SPLINE
SPL {X  -165.650, Y  +532.042, Z    +0.000, E1   +53.611, E3 +284862.764}
SPL {X  -165.650, Y  +526.147, Z    +0.000, E1   +53.495, E3 +284872.403}
SPL {X  -165.650, Y  +517.365, Z    +0.000, E1   +53.387, E3 +284886.571}
SPL {X  -165.650, Y  +505.685, Z    +0.000, E1   +53.701, E3 +284902.196}
SPL {X  -165.650, Y  +498.275, Z    +0.000, E1   +53.357, E3 +284915.504}
SPL {X  -165.650, Y  +487.031, Z    +0.000, E1   +53.931, E3 +284928.912}
SPL {X  -165.650, Y  +450.615, Z    +0.000, E1   +59.721, E3 +284940.152}
SPL {X  -165.650, Y  +449.326, Z    +0.000, E1   +58.606, E3 +284949.202}
SPL {X  -165.650, Y  +442.154, Z    +0.000, E1   +58.369, E3 +284959.826}
SPL {X  -165.650, Y  +437.405, Z    +0.000, E1   +57.663, E3 +284970.435}
SPL {X  -165.650, Y  +432.227, Z    +0.000, E1   +57.103, E3 +284980.923}
SPL {X  -165.650, Y  +428.683, Z    +0.000, E1   +56.222, E3 +284991.277}
SPL {X  -165.650, Y  +424.202, Z    +0.000, E1   +55.382, E3 +285002.966}
SPL {X  -165.650, Y  +418.469, Z    +0.000, E1   +54.594, E3 +285016.074}
SPL {X  -165.650, Y  +413.857, Z    +0.000, E1   +53.683, E3 +285028.645}
SPL {X  -165.650, Y  +403.104, Z    +0.000, E1   +53.908, E3 +285043.382}
SPL {X  -165.650, Y  +393.046, Z    +0.000, E1   +53.951, E3 +285058.066}
SPL {X  -165.650, Y  +383.306, Z    +0.000, E1   +53.987, E3 +285072.343}
SPL {X  -165.640, Y  +376.676, Z    +0.000, E1   +53.760, E3 +285083.510}
SPL {X  -165.408, Y  +369.556, Z    +0.000, E1   +53.942, E3 +285093.061}
SPL {X  -164.927, Y  +363.041, Z    +0.000, E1   +53.687, E3 +285104.356}
SPL {X  -163.980, Y  +355.035, Z    +0.000, E1   +53.657, E3 +285116.553}
SPL {X  -162.665, Y  +347.197, Z    +0.000, E1   +53.396, E3 +285129.816}
SPL {X  -161.218, Y  +340.437, Z    +0.000, E1   +53.207, E3 +285140.915}
SPL {X  -159.523, Y  +333.864, Z    +0.000, E1   +52.908, E3 +285152.537}
SPL {X  -157.624, Y  +327.563, Z    +0.000, E1   +52.705, E3 +285162.946}
SPL {X  -155.665, Y  +321.859, Z    +0.000, E1   +52.064, E3 +285175.119}
SPL {X  -152.682, Y  +314.249, Z    +0.000, E1   +51.841, E3 +285187.567}
SPL {X  -150.607, Y  +309.525, Z    +0.000, E1   +51.147, E3 +285198.052}
SPL {X  -139.567, Y  +289.276, Z    +0.000, E1   +56.334, E3 +285200.030}
SPL {X  -117.053, Y  +261.289, Z    +0.000, E1   +49.815, E3 +285313.564}
ENDSPLINE

SPLINE
SPL {X  -148.836, Y  +305.783, Z    +0.000, E1   +38.029, E3 +285405.041}
SPL {X  -161.816, Y  +343.065, Z    +0.000, E1   +22.147, E3 +285395.691}
SPL {X  -165.007, Y  +363.921, Z    +0.000, E1   +11.079, E3 +285393.680}
SPL {X  -165.587, Y  +373.939, Z    +0.000, E1    +4.928, E3 +285393.520}
SPL {X  -165.650, Y  +378.704, Z    +0.000, E1    +1.700, E3 +285393.101}
SPL {X  -165.650, Y  +382.197, Z    +0.000, E1    -1.038, E3 +285392.175}
SPL {X  -165.650, Y  +386.782, Z    +0.000, E1    -5.783, E3 +285391.652}
SPL {X  -165.650, Y  +392.406, Z    +0.000, E1   -13.042, E3 +285389.550}
SPL {X  -165.650, Y  +398.038, Z    +0.000, E1   -20.113, E3 +285391.117}
SPL {X  -165.650, Y  +403.005, Z    +0.000, E1   -26.762, E3 +285390.299}
SPL {X  -165.650, Y  +415.469, Z    +0.000, E1   -43.461, E3 +285385.122}
SPL {X  -165.650, Y  +460.095, Z    +0.000, E1   -60.221, E3 +285403.383}
SPL {X  -165.650, Y  +535.749, Z    +0.000, E1   -60.559, E3 +285474.227}
ENDSPLINE

SPLINE
SPL {X  -165.650, Y  +516.866, Z    +0.000, E1   -54.768, E3 +285486.777}
ENDSPLINE

SPLINE
SPL {X  -165.650, Y  +521.328, Z    +0.000, E1   -53.870, E3 +285499.068}
SPL {X  -165.650, Y  +531.171, Z    +0.000, E1   -54.075, E3 +285512.413}
SPL {X  -165.650, Y  +538.771, Z    +0.000, E1   -53.840, E3 +285525.153}
SPL {X  -165.650, Y  +545.884, Z    +0.000, E1   -53.883, E3 +285535.458}
SPL {X  -165.650, Y  +553.081, Z    +0.000, E1   -53.834, E3 +285546.591}
SPL {X  -165.650, Y  +560.989, Z    +0.000, E1   -53.974, E3 +285557.428}
SPL {X  -165.650, Y  +568.053, Z    +0.000, E1   -54.124, E3 +285567.018}
SPL {X  -165.650, Y  +577.021, Z    +0.000, E1   -53.813, E3 +285582.517}
SPL {X  -165.650, Y  +587.996, Z    +0.000, E1   -53.969, E3 +285597.754}
SPL {X  -165.650, Y  +595.185, Z    +0.000, E1   -53.962, E3 +285608.464}
SPL {X  -165.650, Y  +602.138, Z    +0.000, E1   -53.941, E3 +285618.958}
SPL {X  -165.650, Y  +610.307, Z    +0.000, E1   -53.995, E3 +285630.806}
SPL {X  -165.650, Y  +617.878, Z    +0.000, E1   -53.838, E3 +285643.062}
SPL {X  -165.650, Y  +626.374, Z    +0.000, E1   -54.092, E3 +285654.078}
SPL {X  -165.650, Y  +632.964, Z    +0.000, E1   -53.887, E3 +285665.205}
SPL {X  -165.650, Y  +643.032, Z    +0.000, E1   -53.946, E3 +285679.950}
SPL {X  -165.650, Y  +654.069, Z    +0.000, E1   -54.108, E3 +285695.309}
SPL {X  -165.650, Y  +659.513, Z    +0.000, E1   -53.578, E3 +285706.536}
SPL {X  -165.650, Y  +667.820, Z    +0.000, E1   -53.975, E3 +285716.601}
SPL {X  -165.650, Y  +674.957, Z    +0.000, E1   -53.977, E3 +285727.113}
SPL {X  -165.574, Y  +680.515, Z    +0.000, E1   -53.820, E3 +285736.440}
SPL {X  -165.171, Y  +688.090, Z    +0.000, E1   -54.025, E3 +285746.400}
SPL {X  -164.558, Y  +694.489, Z    +0.000, E1   -53.745, E3 +285757.750}
SPL {X  -163.580, Y  +701.606, Z    +0.000, E1   -53.591, E3 +285769.183}
SPL {X  -162.702, Y  +706.614, Z    +0.000, E1   -53.230, E3 +285778.849}
SPL {X  -160.941, Y  +714.715, Z    +0.000, E1   -53.321, E3 +285790.469}
SPL {X  -159.638, Y  +719.723, Z    +0.000, E1   -52.685, E3 +285801.471}
SPL {X  -157.868, Y  +725.674, Z    +0.000, E1   -52.862, E3 +285809.328}
SPL {X  -156.314, Y  +730.327, Z    +0.000, E1   -52.199, E3 +285820.010}
SPL {X  -153.975, Y  +736.588, Z    +0.000, E1   -51.877, E3 +285831.040}
SPL {X  -151.949, Y  +741.465, Z    +0.000, E1   -51.645, E3 +285839.445}
SPL {X  -149.075, Y  +747.727, Z    +0.000, E1   -52.134, E3 +285846.160}
SPL {X  -137.775, Y  +767.467, Z    +0.000, E1   -56.912, E3 +285848.823}
SPL {X  -128.847, Y  +779.607, Z    +0.000, E1   -49.118, E3 +285923.840}
SPL {X   -94.133, Y  +811.804, Z    +0.000, E1   -53.019, E3 +285978.474}
ENDSPLINE

SPLINE
SPL {X  -134.098, Y  +772.750, Z    +0.000, E1   -45.587, E3 +286053.768}
SPL {X  -155.319, Y  +733.085, Z    +0.000, E1   -31.947, E3 +286044.646}
SPL {X  -162.077, Y  +709.719, Z    +0.000, E1   -21.590, E3 +286046.324}
SPL {X  -164.499, Y  +694.994, Z    +0.000, E1   -13.860, E3 +286047.108}
SPL {X  -165.513, Y  +682.236, Z    +0.000, E1    -6.385, E3 +286045.444}
SPL {X  -165.650, Y  +675.776, Z    +0.000, E1    -2.014, E3 +286044.752}
SPL {X  -165.650, Y  +672.041, Z    +0.000, E1    +0.844, E3 +286043.700}
SPL {X  -165.650, Y  +667.328, Z    +0.000, E1    +5.806, E3 +286043.076}
SPL {X  -165.650, Y  +661.774, Z    +0.000, E1   +13.006, E3 +286041.400}
SPL {X  -165.650, Y  +654.085, Z    +0.000, E1   +23.232, E3 +286041.260}
SPL {X  -165.650, Y  +639.700, Z    +0.000, E1   +43.326, E3 +286035.387}
SPL {X  -165.650, Y  +605.320, Z    +0.000, E1   +76.562, E3 +286014.796}
SPL {X  -165.650, Y  +596.505, Z    +0.000, E1   +55.802, E3 +286064.152}
SPL {X  -165.650, Y  +521.429, Z    +0.000, E1   +61.144, E3 +286119.637}
ENDSPLINE

SPLINE
SPL {X  -165.650, Y  +526.028, Z    +0.000, E1   +58.071, E3 +286133.411}
SPL {X  -165.650, Y  +539.856, Z    +0.000, E1   +53.398, E3 +286143.959}
ENDSPLINE

SPLINE
SPL {X  -165.650, Y  +532.042, Z    +0.000, E1   +53.611, E3 +286154.430}
SPL {X  -165.650, Y  +526.147, Z    +0.000, E1   +53.495, E3 +286164.069}
SPL {X  -165.650, Y  +517.365, Z    +0.000, E1   +53.387, E3 +286178.237}
SPL {X  -165.650, Y  +505.685, Z    +0.000, E1   +53.701, E3 +286193.863}
SPL {X  -165.650, Y  +498.275, Z    +0.000, E1   +53.357, E3 +286207.170}
SPL {X  -165.650, Y  +487.031, Z    +0.000, E1   +53.931, E3 +286220.579}
SPL {X  -165.650, Y  +450.615, Z    +0.000, E1   +59.721, E3 +286231.819}
SPL {X  -165.650, Y  +449.326, Z    +0.000, E1   +58.606, E3 +286240.868}
SPL {X  -165.650, Y  +442.154, Z    +0.000, E1   +58.369, E3 +286251.492}
SPL {X  -165.650, Y  +437.405, Z    +0.000, E1   +57.663, E3 +286262.102}
SPL {X  -165.650, Y  +432.227, Z    +0.000, E1   +57.103, E3 +286272.590}
SPL {X  -165.650, Y  +428.683, Z    +0.000, E1   +56.222, E3 +286282.944}
SPL {X  -165.650, Y  +424.202, Z    +0.000, E1   +55.382, E3 +286294.633}
SPL {X  -165.650, Y  +418.756, Z    +0.000, E1   +54.154, E3 +286310.312}
SPL {X  -165.650, Y  +410.508, Z    +0.000, E1   +54.007, E3 +286323.267}
SPL {X  -165.650, Y  +403.104, Z    +0.000, E1   +53.908, E3 +286335.049}
SPL {X  -165.650, Y  +391.401, Z    +0.000, E1   +53.934, E3 +286352.440}
SPL {X  -165.650, Y  +378.987, Z    +0.000, E1   +53.974, E3 +286370.636}
SPL {X  -165.408, Y  +369.556, Z    +0.000, E1   +53.942, E3 +286384.727}
SPL {X  -164.927, Y  +363.041, Z    +0.000, E1   +53.687, E3 +286396.023}
SPL {X  -164.096, Y  +355.862, Z    +0.000, E1   +53.838, E3 +286405.753}
SPL {X  -163.142, Y  +349.785, Z    +0.000, E1   +53.493, E3 +286416.969}
SPL {X  -161.604, Y  +342.113, Z    +0.000, E1   +53.155, E3 +286430.463}
SPL {X  -160.424, Y  +337.221, Z    +0.000, E1   +52.694, E3 +286440.303}
SPL {X  -158.192, Y  +329.354, Z    +0.000, E1   +52.890, E3 +286451.135}
SPL {X  -155.665, Y  +321.859, Z    +0.000, E1   +52.064, E3 +286466.786}
SPL {X  -152.682, Y  +314.249, Z    +0.000, E1   +51.841, E3 +286479.234}
SPL {X  -150.607, Y  +309.525, Z    +0.000, E1   +51.147, E3 +286489.719}
SPL {X  -139.567, Y  +289.276, Z    +0.000, E1   +56.334, E3 +286491.697}
SPL {X  -117.053, Y  +261.289, Z    +0.000, E1   +49.815, E3 +286605.230}
ENDSPLINE

SPLINE
SPL {X  -148.836, Y  +305.783, Z    +0.000, E1   +38.029, E3 +286696.708}
SPL {X  -161.816, Y  +343.065, Z    +0.000, E1   +22.147, E3 +286687.358}
SPL {X  -164.614, Y  +360.007, Z    +0.000, E1   +13.213, E3 +286683.144}
SPL {X  -165.520, Y  +371.933, Z    +0.000, E1    +6.276, E3 +286685.899}
SPL {X  -165.650, Y  +378.704, Z    +0.000, E1    +1.700, E3 +286684.768}
SPL {X  -165.650, Y  +382.197, Z    +0.000, E1    -1.038, E3 +286683.841}
SPL {X  -165.650, Y  +386.782, Z    +0.000, E1    -5.783, E3 +286683.319}
SPL {X  -165.650, Y  +392.406, Z    +0.000, E1   -13.042, E3 +286681.216}
SPL {X  -165.650, Y  +400.489, Z    +0.000, E1   -23.243, E3 +286682.380}
SPL {X  -165.650, Y  +415.469, Z    +0.000, E1   -43.461, E3 +286676.789}
SPL {X  -165.650, Y  +460.095, Z    +0.000, E1   -60.221, E3 +286695.050}
SPL {X  -165.650, Y  +535.749, Z    +0.000, E1   -60.559, E3 +286765.894}
ENDSPLINE

SPLINE
SPL {X  -165.650, Y  +516.866, Z    +0.000, E1   -54.768, E3 +286778.444}
ENDSPLINE

SPLINE
SPL {X  -165.650, Y  +521.328, Z    +0.000, E1   -53.870, E3 +286790.735}
SPL {X  -165.650, Y  +531.171, Z    +0.000, E1   -54.075, E3 +286804.079}
SPL {X  -165.650, Y  +538.771, Z    +0.000, E1   -53.840, E3 +286816.820}
SPL {X  -165.650, Y  +545.884, Z    +0.000, E1   -53.883, E3 +286827.124}
SPL {X  -165.650, Y  +553.081, Z    +0.000, E1   -53.834, E3 +286838.257}
SPL {X  -165.650, Y  +560.989, Z    +0.000, E1   -53.974, E3 +286849.094}
SPL {X  -165.650, Y  +568.053, Z    +0.000, E1   -54.124, E3 +286858.685}
SPL {X  -165.650, Y  +577.021, Z    +0.000, E1   -53.813, E3 +286874.183}
SPL {X  -165.650, Y  +587.996, Z    +0.000, E1   -53.969, E3 +286889.421}
SPL {X  -165.650, Y  +595.185, Z    +0.000, E1   -53.962, E3 +286900.130}
SPL {X  -165.650, Y  +602.138, Z    +0.000, E1   -53.941, E3 +286910.625}
SPL {X  -165.650, Y  +610.307, Z    +0.000, E1   -53.995, E3 +286922.472}
SPL {X  -165.650, Y  +617.878, Z    +0.000, E1   -53.838, E3 +286934.729}
SPL {X  -165.650, Y  +627.853, Z    +0.000, E1   -53.937, E3 +286949.083}
SPL {X  -165.650, Y  +638.510, Z    +0.000, E1   -54.057, E3 +286964.142}
SPL {X  -165.650, Y  +645.417, Z    +0.000, E1   -53.856, E3 +286975.556}
SPL {X  -165.650, Y  +654.069, Z    +0.000, E1   -54.108, E3 +286986.976}
SPL {X  -165.650, Y  +659.513, Z    +0.000, E1   -53.578, E3 +286998.203}
SPL {X  -165.650, Y  +667.820, Z    +0.000, E1   -53.975, E3 +287008.268}
SPL {X  -165.650, Y  +674.957, Z    +0.000, E1   -53.977, E3 +287018.780}
SPL {X  -165.574, Y  +680.515, Z    +0.000, E1   -53.820, E3 +287028.107}
SPL {X  -165.171, Y  +688.090, Z    +0.000, E1   -54.025, E3 +287038.067}
SPL {X  -164.558, Y  +694.489, Z    +0.000, E1   -53.745, E3 +287049.416}
SPL {X  -163.580, Y  +701.606, Z    +0.000, E1   -53.591, E3 +287060.849}
SPL {X  -162.702, Y  +706.614, Z    +0.000, E1   -53.230, E3 +287070.516}
SPL {X  -161.265, Y  +713.361, Z    +0.000, E1   -53.436, E3 +287079.325}
SPL {X  -159.936, Y  +718.632, Z    +0.000, E1   -52.857, E3 +287090.654}
SPL {X  -157.868, Y  +725.674, Z    +0.000, E1   -52.862, E3 +287100.995}
SPL {X  -156.314, Y  +730.327, Z    +0.000, E1   -52.199, E3 +287111.676}
SPL {X  -153.975, Y  +736.588, Z    +0.000, E1   -51.877, E3 +287122.707}
SPL {X  -151.949, Y  +741.465, Z    +0.000, E1   -51.645, E3 +287131.112}
SPL {X  -149.075, Y  +747.727, Z    +0.000, E1   -52.134, E3 +287137.827}
SPL {X  -137.775, Y  +767.467, Z    +0.000, E1   -56.912, E3 +287140.490}
SPL {X  -128.847, Y  +779.607, Z    +0.000, E1   -49.118, E3 +287215.506}
SPL {X   -94.133, Y  +811.804, Z    +0.000, E1   -53.019, E3 +287270.141}
ENDSPLINE

SPLINE
SPL {X  -134.098, Y  +772.750, Z    +0.000, E1   -45.587, E3 +287345.435}
SPL {X  -155.319, Y  +733.085, Z    +0.000, E1   -31.947, E3 +287336.313}
SPL {X  -162.077, Y  +709.719, Z    +0.000, E1   -21.590, E3 +287337.990}
SPL {X  -164.499, Y  +694.994, Z    +0.000, E1   -13.860, E3 +287338.775}
SPL {X  -165.382, Y  +684.927, Z    +0.000, E1    -7.984, E3 +287336.952}
SPL {X  -165.645, Y  +676.778, Z    +0.000, E1    -2.777, E3 +287336.675}
SPL {X  -165.650, Y  +672.041, Z    +0.000, E1    +0.844, E3 +287335.366}
SPL {X  -165.650, Y  +667.328, Z    +0.000, E1    +5.806, E3 +287334.743}
SPL {X  -165.650, Y  +661.774, Z    +0.000, E1   +13.006, E3 +287333.067}
SPL {X  -165.650, Y  +656.573, Z    +0.000, E1   +19.875, E3 +287333.626}
SPL {X  -165.650, Y  +650.769, Z    +0.000, E1   +28.083, E3 +287331.992}
SPL {X  -165.650, Y  +639.700, Z    +0.000, E1   +43.326, E3 +287327.054}
SPL {X  -165.650, Y  +605.320, Z    +0.000, E1   +76.562, E3 +287306.463}
SPL {X  -165.650, Y  +597.745, Z    +0.000, E1   +59.636, E3 +287344.464}
SPL {X  -165.650, Y  +596.360, Z    +0.000, E1   +54.978, E3 +287358.072}
SPL {X  -165.650, Y  +521.429, Z    +0.000, E1   +61.144, E3 +287411.303}
ENDSPLINE

SPLINE
SPL {X  -165.650, Y  +526.028, Z    +0.000, E1   +58.071, E3 +287425.078}
SPL {X  -165.650, Y  +539.856, Z    +0.000, E1   +53.398, E3 +287435.626}
ENDSPLINE

SPLINE
SPL {X  -165.650, Y  +532.042, Z    +0.000, E1   +53.611, E3 +287446.097}
SPL {X  -165.650, Y  +526.147, Z    +0.000, E1   +53.495, E3 +287455.736}
SPL {X  -165.650, Y  +517.365, Z    +0.000, E1   +53.387, E3 +287469.904}
SPL {X  -165.650, Y  +505.685, Z    +0.000, E1   +53.701, E3 +287485.529}
SPL {X  -165.650, Y  +498.275, Z    +0.000, E1   +53.357, E3 +287498.837}
SPL {X  -165.650, Y  +487.031, Z    +0.000, E1   +53.931, E3 +287512.246}
SPL {X  -165.650, Y  +450.615, Z    +0.000, E1   +59.721, E3 +287523.486}
SPL {X  -165.650, Y  +449.326, Z    +0.000, E1   +58.606, E3 +287532.535}
SPL {X  -165.650, Y  +442.154, Z    +0.000, E1   +58.369, E3 +287543.159}
SPL {X  -165.650, Y  +437.405, Z    +0.000, E1   +57.663, E3 +287553.769}
SPL {X  -165.650, Y  +432.227, Z    +0.000, E1   +57.103, E3 +287564.256}
SPL {X  -165.650, Y  +428.683, Z    +0.000, E1   +56.222, E3 +287574.611}
SPL {X  -165.650, Y  +424.202, Z    +0.000, E1   +55.382, E3 +287586.300}
SPL {X  -165.650, Y  +418.469, Z    +0.000, E1   +54.594, E3 +287599.408}
SPL {X  -165.650, Y  +413.857, Z    +0.000, E1   +53.683, E3 +287611.979}
SPL {X  -165.650, Y  +403.104, Z    +0.000, E1   +53.908, E3 +287626.716}
SPL {X  -165.650, Y  +391.401, Z    +0.000, E1   +53.934, E3 +287644.106}
SPL {X  -165.650, Y  +378.987, Z    +0.000, E1   +53.974, E3 +287662.303}
SPL {X  -165.408, Y  +369.556, Z    +0.000, E1   +53.942, E3 +287676.394}
SPL {X  -164.927, Y  +363.041, Z    +0.000, E1   +53.687, E3 +287687.690}
SPL {X  -164.096, Y  +355.862, Z    +0.000, E1   +53.838, E3 +287697.420}
SPL {X  -163.142, Y  +349.785, Z    +0.000, E1   +53.493, E3 +287708.636}
SPL {X  -161.604, Y  +342.113, Z    +0.000, E1   +53.155, E3 +287722.130}
SPL {X  -159.523, Y  +333.864, Z    +0.000, E1   +52.908, E3 +287735.870}
SPL {X  -157.624, Y  +327.563, Z    +0.000, E1   +52.705, E3 +287746.280}
SPL {X  -156.289, Y  +323.602, Z    +0.000, E1   +52.159, E3 +287755.168}
SPL {X  -154.898, Y  +319.792, Z    +0.000, E1   +51.850, E3 +287762.504}
SPL {X  -152.682, Y  +314.249, Z    +0.000, E1   +51.841, E3 +287770.901}
SPL {X  -150.607, Y  +309.525, Z    +0.000, E1   +51.147, E3 +287781.385}
SPL {X  -139.567, Y  +289.276, Z    +0.000, E1   +56.334, E3 +287783.363}
SPL {X  -117.053, Y  +261.289, Z    +0.000, E1   +49.815, E3 +287896.897}
ENDSPLINE

SPLINE
SPL {X  -148.836, Y  +305.783, Z    +0.000, E1   +38.029, E3 +287988.375}
SPL {X  -161.816, Y  +343.065, Z    +0.000, E1   +22.147, E3 +287979.025}
SPL {X  -164.614, Y  +360.007, Z    +0.000, E1   +13.213, E3 +287974.811}
SPL {X  -165.520, Y  +371.933, Z    +0.000, E1    +6.276, E3 +287977.565}
SPL {X  -165.650, Y  +380.164, Z    +0.000, E1    +0.707, E3 +287976.035}
SPL {X  -165.650, Y  +384.850, Z    +0.000, E1    -3.598, E3 +287975.142}
SPL {X  -165.650, Y  +391.255, Z    +0.000, E1   -11.346, E3 +287973.484}
SPL {X  -165.650, Y  +398.038, Z    +0.000, E1   -20.113, E3 +287974.450}
SPL {X  -165.650, Y  +403.005, Z    +0.000, E1   -26.762, E3 +287973.632}
SPL {X  -165.650, Y  +415.469, Z    +0.000, E1   -43.461, E3 +287968.455}
SPL {X  -165.650, Y  +460.095, Z    +0.000, E1   -60.221, E3 +287986.717}
SPL {X  -165.650, Y  +535.749, Z    +0.000, E1   -60.559, E3 +288057.560}
ENDSPLINE

SPLINE
SPL {X  -165.650, Y  +516.866, Z    +0.000, E1   -54.768, E3 +288070.110}
ENDSPLINE

SPLINE
SPL {X  -165.650, Y  +521.328, Z    +0.000, E1   -53.870, E3 +288082.402}
SPL {X  -165.650, Y  +531.171, Z    +0.000, E1   -54.075, E3 +288095.746}
SPL {X  -165.650, Y  +538.771, Z    +0.000, E1   -53.840, E3 +288108.486}
SPL {X  -165.650, Y  +545.884, Z    +0.000, E1   -53.883, E3 +288118.791}
SPL {X  -165.650, Y  +553.081, Z    +0.000, E1   -53.834, E3 +288129.924}
SPL {X  -165.650, Y  +560.989, Z    +0.000, E1   -53.974, E3 +288140.761}
SPL {X  -165.650, Y  +568.053, Z    +0.000, E1   -54.124, E3 +288150.351}
SPL {X  -165.650, Y  +577.021, Z    +0.000, E1   -53.813, E3 +288165.850}
SPL {X  -165.650, Y  +587.996, Z    +0.000, E1   -53.969, E3 +288181.088}
SPL {X  -165.650, Y  +595.185, Z    +0.000, E1   -53.962, E3 +288191.797}
SPL {X  -165.650, Y  +602.138, Z    +0.000, E1   -53.941, E3 +288202.291}
SPL {X  -165.650, Y  +610.307, Z    +0.000, E1   -53.995, E3 +288214.139}
SPL {X  -165.650, Y  +617.878, Z    +0.000, E1   -53.838, E3 +288226.396}
SPL {X  -165.650, Y  +627.853, Z    +0.000, E1   -53.937, E3 +288240.749}
SPL {X  -165.650, Y  +638.510, Z    +0.000, E1   -54.057, E3 +288255.809}
SPL {X  -165.650, Y  +647.911, Z    +0.000, E1   -53.930, E3 +288270.608}
SPL {X  -165.650, Y  +656.836, Z    +0.000, E1   -54.184, E3 +288282.140}
SPL {X  -165.650, Y  +659.513, Z    +0.000, E1   -53.578, E3 +288289.869}
SPL {X  -165.650, Y  +667.820, Z    +0.000, E1   -53.975, E3 +288299.934}
SPL {X  -165.623, Y  +678.503, Z    +0.000, E1   -53.932, E3 +288316.286}
SPL {X  -165.171, Y  +688.090, Z    +0.000, E1   -54.025, E3 +288329.734}
SPL {X  -164.558, Y  +694.489, Z    +0.000, E1   -53.745, E3 +288341.083}
SPL {X  -163.580, Y  +701.606, Z    +0.000, E1   -53.591, E3 +288352.516}
SPL {X  -162.702, Y  +706.614, Z    +0.000, E1   -53.230, E3 +288362.183}
SPL {X  -160.941, Y  +714.715, Z    +0.000, E1   -53.321, E3 +288373.802}
SPL {X  -159.638, Y  +719.723, Z    +0.000, E1   -52.685, E3 +288384.805}
SPL {X  -157.521, Y  +726.754, Z    +0.000, E1   -52.585, E3 +288396.000}
SPL {X  -155.632, Y  +732.234, Z    +0.000, E1   -52.209, E3 +288406.047}
SPL {X  -153.975, Y  +736.588, Z    +0.000, E1   -51.877, E3 +288414.373}
SPL {X  -151.949, Y  +741.465, Z    +0.000, E1   -51.645, E3 +288422.779}
SPL {X  -149.075, Y  +747.727, Z    +0.000, E1   -52.134, E3 +288429.493}
SPL {X  -137.775, Y  +767.467, Z    +0.000, E1   -56.912, E3 +288432.157}
SPL {X  -128.847, Y  +779.607, Z    +0.000, E1   -49.118, E3 +288507.173}
SPL {X   -94.133, Y  +811.804, Z    +0.000, E1   -53.019, E3 +288561.807}
ENDSPLINE

SPLINE
SPL {X  -134.098, Y  +772.750, Z    +0.000, E1   -45.587, E3 +288637.102}
SPL {X  -155.319, Y  +733.085, Z    +0.000, E1   -31.947, E3 +288627.979}
SPL {X  -162.077, Y  +709.719, Z    +0.000, E1   -21.590, E3 +288629.657}
SPL {X  -164.499, Y  +694.994, Z    +0.000, E1   -13.860, E3 +288630.442}
SPL {X  -165.382, Y  +684.927, Z    +0.000, E1    -7.984, E3 +288628.619}
SPL {X  -165.645, Y  +676.778, Z    +0.000, E1    -2.777, E3 +288628.341}
SPL {X  -165.650, Y  +672.041, Z    +0.000, E1    +0.844, E3 +288627.033}
SPL {X  -165.650, Y  +667.328, Z    +0.000, E1    +5.806, E3 +288626.410}
SPL {X  -165.650, Y  +661.774, Z    +0.000, E1   +13.006, E3 +288624.734}
SPL {X  -165.650, Y  +656.573, Z    +0.000, E1   +19.875, E3 +288625.292}
SPL {X  -165.650, Y  +650.769, Z    +0.000, E1   +28.083, E3 +288623.658}
SPL {X  -165.650, Y  +639.700, Z    +0.000, E1   +43.326, E3 +288618.720}
SPL {X  -165.650, Y  +605.320, Z    +0.000, E1   +76.562, E3 +288598.130}
SPL {X  -165.650, Y  +597.745, Z    +0.000, E1   +59.636, E3 +288636.131}
SPL {X  -165.650, Y  +596.360, Z    +0.000, E1   +54.978, E3 +288649.739}
SPL {X  -165.650, Y  +521.429, Z    +0.000, E1   +61.144, E3 +288702.970}
ENDSPLINE

SPLINE
SPL {X  -165.650, Y  +526.028, Z    +0.000, E1   +58.071, E3 +288716.745}
SPL {X  -165.650, Y  +539.856, Z    +0.000, E1   +53.398, E3 +288727.292}
ENDSPLINE

SPLINE
SPL {X  -165.650, Y  +532.042, Z    +0.000, E1   +53.611, E3 +288737.764}
SPL {X  -165.650, Y  +526.147, Z    +0.000, E1   +53.495, E3 +288747.403}
SPL {X  -165.650, Y  +517.365, Z    +0.000, E1   +53.387, E3 +288761.571}
SPL {X  -165.650, Y  +505.685, Z    +0.000, E1   +53.701, E3 +288777.196}
SPL {X  -165.650, Y  +498.275, Z    +0.000, E1   +53.357, E3 +288790.504}
SPL {X  -165.650, Y  +487.031, Z    +0.000, E1   +53.931, E3 +288803.912}
SPL {X  -165.650, Y  +450.615, Z    +0.000, E1   +59.721, E3 +288815.152}
SPL {X  -165.650, Y  +449.326, Z    +0.000, E1   +58.606, E3 +288824.202}
SPL {X  -165.650, Y  +442.154, Z    +0.000, E1   +58.369, E3 +288834.826}
SPL {X  -165.650, Y  +437.405, Z    +0.000, E1   +57.663, E3 +288845.435}
SPL {X  -165.650, Y  +432.227, Z    +0.000, E1   +57.103, E3 +288855.923}
SPL {X  -165.650, Y  +428.683, Z    +0.000, E1   +56.222, E3 +288866.277}
SPL {X  -165.650, Y  +424.202, Z    +0.000, E1   +55.382, E3 +288877.966}
SPL {X  -165.650, Y  +418.469, Z    +0.000, E1   +54.594, E3 +288891.074}
SPL {X  -165.650, Y  +413.857, Z    +0.000, E1   +53.683, E3 +288903.645}
SPL {X  -165.650, Y  +403.104, Z    +0.000, E1   +53.908, E3 +288918.382}
SPL {X  -165.650, Y  +393.046, Z    +0.000, E1   +53.951, E3 +288933.066}
SPL {X  -165.650, Y  +383.306, Z    +0.000, E1   +53.987, E3 +288947.343}
SPL {X  -165.640, Y  +376.676, Z    +0.000, E1   +53.760, E3 +288958.510}
SPL {X  -165.408, Y  +369.556, Z    +0.000, E1   +53.942, E3 +288968.061}
SPL {X  -164.927, Y  +363.041, Z    +0.000, E1   +53.687, E3 +288979.356}
SPL {X  -163.980, Y  +355.035, Z    +0.000, E1   +53.657, E3 +288991.553}
SPL {X  -162.665, Y  +347.197, Z    +0.000, E1   +53.396, E3 +289004.816}
SPL {X  -161.218, Y  +340.437, Z    +0.000, E1   +53.207, E3 +289015.915}
SPL {X  -159.523, Y  +333.864, Z    +0.000, E1   +52.908, E3 +289027.537}
SPL {X  -157.624, Y  +327.563, Z    +0.000, E1   +52.705, E3 +289037.946}
SPL {X  -155.665, Y  +321.859, Z    +0.000, E1   +52.064, E3 +289050.119}
SPL {X  -152.682, Y  +314.249, Z    +0.000, E1   +51.841, E3 +289062.567}
SPL {X  -150.607, Y  +309.525, Z    +0.000, E1   +51.147, E3 +289073.052}
SPL {X  -139.567, Y  +289.276, Z    +0.000, E1   +56.334, E3 +289075.030}
SPL {X  -117.053, Y  +261.289, Z    +0.000, E1   +49.815, E3 +289188.564}
ENDSPLINE

SPLINE
SPL {X  -148.836, Y  +305.783, Z    +0.000, E1   +38.029, E3 +289280.041}
SPL {X  -161.816, Y  +343.065, Z    +0.000, E1   +22.147, E3 +289270.691}
SPL {X  -165.007, Y  +363.921, Z    +0.000, E1   +11.079, E3 +289268.680}
SPL {X  -165.587, Y  +373.939, Z    +0.000, E1    +4.928, E3 +289268.520}
SPL {X  -165.650, Y  +378.704, Z    +0.000, E1    +1.700, E3 +289268.101}
SPL {X  -165.650, Y  +382.197, Z    +0.000, E1    -1.038, E3 +289267.175}
SPL {X  -165.650, Y  +386.782, Z    +0.000, E1    -5.783, E3 +289266.652}
SPL {X  -165.650, Y  +392.406, Z    +0.000, E1   -13.042, E3 +289264.550}
SPL {X  -165.650, Y  +398.038, Z    +0.000, E1   -20.113, E3 +289266.117}
SPL {X  -165.650, Y  +403.005, Z    +0.000, E1   -26.762, E3 +289265.299}
SPL {X  -165.650, Y  +415.469, Z    +0.000, E1   -43.461, E3 +289260.122}
SPL {X  -165.650, Y  +460.095, Z    +0.000, E1   -60.221, E3 +289278.383}
SPL {X  -165.650, Y  +535.749, Z    +0.000, E1   -60.559, E3 +289349.227}
ENDSPLINE

SPLINE
SPL {X  -165.650, Y  +516.866, Z    +0.000, E1   -54.768, E3 +289361.777}
ENDSPLINE

SPLINE
SPL {X  -165.650, Y  +521.328, Z    +0.000, E1   -53.870, E3 +289374.068}
SPL {X  -165.650, Y  +531.171, Z    +0.000, E1   -54.075, E3 +289387.413}
SPL {X  -165.650, Y  +538.771, Z    +0.000, E1   -53.840, E3 +289400.153}
SPL {X  -165.650, Y  +545.884, Z    +0.000, E1   -53.883, E3 +289410.458}
SPL {X  -165.650, Y  +553.081, Z    +0.000, E1   -53.834, E3 +289421.591}
SPL {X  -165.650, Y  +560.989, Z    +0.000, E1   -53.974, E3 +289432.428}
SPL {X  -165.650, Y  +568.053, Z    +0.000, E1   -54.124, E3 +289442.018}
SPL {X  -165.650, Y  +577.021, Z    +0.000, E1   -53.813, E3 +289457.517}
SPL {X  -165.650, Y  +587.996, Z    +0.000, E1   -53.969, E3 +289472.754}
SPL {X  -165.650, Y  +595.185, Z    +0.000, E1   -53.962, E3 +289483.464}
SPL {X  -165.650, Y  +602.138, Z    +0.000, E1   -53.941, E3 +289493.958}
SPL {X  -165.650, Y  +610.307, Z    +0.000, E1   -53.995, E3 +289505.806}
SPL {X  -165.650, Y  +617.878, Z    +0.000, E1   -53.838, E3 +289518.062}
SPL {X  -165.650, Y  +626.374, Z    +0.000, E1   -54.092, E3 +289529.078}
SPL {X  -165.650, Y  +632.964, Z    +0.000, E1   -53.887, E3 +289540.205}
SPL {X  -165.650, Y  +643.032, Z    +0.000, E1   -53.946, E3 +289554.950}
SPL {X  -165.650, Y  +654.069, Z    +0.000, E1   -54.108, E3 +289570.309}
SPL {X  -165.650, Y  +659.513, Z    +0.000, E1   -53.578, E3 +289581.536}
SPL {X  -165.650, Y  +667.820, Z    +0.000, E1   -53.975, E3 +289591.601}
SPL {X  -165.650, Y  +674.957, Z    +0.000, E1   -53.977, E3 +289602.113}
SPL {X  -165.574, Y  +680.515, Z    +0.000, E1   -53.820, E3 +289611.440}
SPL {X  -165.171, Y  +688.090, Z    +0.000, E1   -54.025, E3 +289621.400}
SPL {X  -164.558, Y  +694.489, Z    +0.000, E1   -53.745, E3 +289632.750}
SPL {X  -163.580, Y  +701.606, Z    +0.000, E1   -53.591, E3 +289644.183}
SPL {X  -162.702, Y  +706.614, Z    +0.000, E1   -53.230, E3 +289653.849}
SPL {X  -160.941, Y  +714.715, Z    +0.000, E1   -53.321, E3 +289665.469}
SPL {X  -159.638, Y  +719.723, Z    +0.000, E1   -52.685, E3 +289676.471}
SPL {X  -157.868, Y  +725.674, Z    +0.000, E1   -52.862, E3 +289684.328}
SPL {X  -156.314, Y  +730.327, Z    +0.000, E1   -52.199, E3 +289695.010}
SPL {X  -153.975, Y  +736.588, Z    +0.000, E1   -51.877, E3 +289706.040}
SPL {X  -151.949, Y  +741.465, Z    +0.000, E1   -51.645, E3 +289714.445}
SPL {X  -149.075, Y  +747.727, Z    +0.000, E1   -52.134, E3 +289721.160}
SPL {X  -137.775, Y  +767.467, Z    +0.000, E1   -56.912, E3 +289723.823}
SPL {X  -128.847, Y  +779.607, Z    +0.000, E1   -49.118, E3 +289798.840}
SPL {X   -94.133, Y  +811.804, Z    +0.000, E1   -53.019, E3 +289853.474}
ENDSPLINE

SPLINE
SPL {X  -134.098, Y  +772.750, Z    +0.000, E1   -45.587, E3 +289928.768}
SPL {X  -155.319, Y  +733.085, Z    +0.000, E1   -31.947, E3 +289919.646}
SPL {X  -162.077, Y  +709.719, Z    +0.000, E1   -21.590, E3 +289921.324}
SPL {X  -164.499, Y  +694.994, Z    +0.000, E1   -13.860, E3 +289922.108}
SPL {X  -165.382, Y  +684.927, Z    +0.000, E1    -7.984, E3 +289920.286}
SPL {X  -165.645, Y  +676.778, Z    +0.000, E1    -2.777, E3 +289920.008}
SPL {X  -165.650, Y  +672.938, Z    +0.000, E1    +0.157, E3 +289918.767}
SPL {X  -165.650, Y  +669.402, Z    +0.000, E1    +3.448, E3 +289918.158}
SPL {X  -165.650, Y  +663.061, Z    +0.000, E1   +11.076, E3 +289917.152}
SPL {X  -165.650, Y  +656.573, Z    +0.000, E1   +19.875, E3 +289916.959}
SPL {X  -165.650, Y  +647.335, Z    +0.000, E1   +32.835, E3 +289913.881}
SPL {X  -165.650, Y  +637.438, Z    +0.000, E1   +46.409, E3 +289909.241}
SPL {X  -165.650, Y  +605.320, Z    +0.000, E1   +76.562, E3 +289889.796}
SPL {X  -165.650, Y  +596.505, Z    +0.000, E1   +55.802, E3 +289939.152}
SPL {X  -165.650, Y  +524.050, Z    +0.000, E1   +59.300, E3 +290003.312}
ENDSPLINE

SPLINE
SPL {X  -165.650, Y  +539.856, Z    +0.000, E1   +53.398, E3 +290018.959}
ENDSPLINE

SPLINE
SPL {X  -165.650, Y  +530.389, Z    +0.000, E1   +53.621, E3 +290031.964}
SPL {X  -165.650, Y  +521.849, Z    +0.000, E1   +53.452, E3 +290045.904}
SPL {X  -165.650, Y  +512.447, Z    +0.000, E1   +53.456, E3 +290060.163}
SPL {X  -165.650, Y  +503.994, Z    +0.000, E1   +53.652, E3 +290071.602}
SPL {X  -165.650, Y  +498.275, Z    +0.000, E1   +53.357, E3 +290082.170}
SPL {X  -165.650, Y  +487.031, Z    +0.000, E1   +53.931, E3 +290095.579}
SPL {X  -165.650, Y  +450.615, Z    +0.000, E1   +59.721, E3 +290106.819}
SPL {X  -165.650, Y  +449.326, Z    +0.000, E1   +58.606, E3 +290115.868}
SPL {X  -165.650, Y  +442.154, Z    +0.000, E1   +58.369, E3 +290126.492}
SPL {X  -165.650, Y  +437.405, Z    +0.000, E1   +57.663, E3 +290137.102}
SPL {X  -165.650, Y  +432.227, Z    +0.000, E1   +57.103, E3 +290147.590}
SPL {X  -165.650, Y  +428.683, Z    +0.000, E1   +56.222, E3 +290157.944}
SPL {X  -165.650, Y  +424.202, Z    +0.000, E1   +55.382, E3 +290169.633}
SPL {X  -165.650, Y  +420.516, Z    +0.000, E1   +54.144, E3 +290182.638}
SPL {X  -165.650, Y  +412.197, Z    +0.000, E1   +54.057, E3 +290195.560}
SPL {X  -165.650, Y  +405.379, Z    +0.000, E1   +53.922, E3 +290206.426}
SPL {X  -165.650, Y  +400.791, Z    +0.000, E1   +53.827, E3 +290213.840}
SPL {X  -165.650, Y  +391.401, Z    +0.000, E1   +53.934, E3 +290227.440}
SPL {X  -165.650, Y  +381.191, Z    +0.000, E1   +54.078, E3 +290241.510}
SPL {X  -165.600, Y  +374.450, Z    +0.000, E1   +53.824, E3 +290253.211}
SPL {X  -165.050, Y  +364.408, Z    +0.000, E1   +53.830, E3 +290268.270}
SPL {X  -164.096, Y  +355.862, Z    +0.000, E1   +53.838, E3 +290280.753}
SPL {X  -162.936, Y  +348.637, Z    +0.000, E1   +53.390, E3 +290294.469}
SPL {X  -161.218, Y  +340.437, Z    +0.000, E1   +53.207, E3 +290307.581}
SPL {X  -159.523, Y  +333.864, Z    +0.000, E1   +52.908, E3 +290319.204}
SPL {X  -157.624, Y  +327.563, Z    +0.000, E1   +52.705, E3 +290329.613}
SPL {X  -155.665, Y  +321.859, Z    +0.000, E1   +52.064, E3 +290341.786}
SPL {X  -152.682, Y  +314.249, Z    +0.000, E1   +51.841, E3 +290354.234}
SPL {X  -150.607, Y  +309.525, Z    +0.000, E1   +51.147, E3 +290364.719}
SPL {X  -139.567, Y  +289.276, Z    +0.000, E1   +56.334, E3 +290366.697}
SPL {X  -117.053, Y  +261.289, Z    +0.000, E1   +49.815, E3 +290480.230}
ENDSPLINE

SPLINE
SPL {X  -148.836, Y  +305.783, Z    +0.000, E1   +38.029, E3 +290571.708}
SPL {X  -161.816, Y  +343.065, Z    +0.000, E1   +22.147, E3 +290562.358}
SPL {X  -164.614, Y  +360.007, Z    +0.000, E1   +13.213, E3 +290558.144}
SPL {X  -165.520, Y  +371.933, Z    +0.000, E1    +6.276, E3 +290560.899}
SPL {X  -165.650, Y  +378.704, Z    +0.000, E1    +1.700, E3 +290559.768}
SPL {X  -165.650, Y  +382.197, Z    +0.000, E1    -1.038, E3 +290558.841}
SPL {X  -165.650, Y  +386.782, Z    +0.000, E1    -5.783, E3 +290558.319}
SPL {X  -165.650, Y  +392.406, Z    +0.000, E1   -13.042, E3 +290556.216}
SPL {X  -165.650, Y  +400.489, Z    +0.000, E1   -23.243, E3 +290557.380}
SPL {X  -165.650, Y  +415.469, Z    +0.000, E1   -43.461, E3 +290551.789}
SPL {X  -165.650, Y  +460.095, Z    +0.000, E1   -60.221, E3 +290570.050}
SPL {X  -165.650, Y  +535.749, Z    +0.000, E1   -60.559, E3 +290640.894}
ENDSPLINE

SPLINE
SPL {X  -165.650, Y  +516.750, Z    +0.000, E1   -54.244, E3 +290656.744}
ENDSPLINE

SPLINE
SPL {X  -165.650, Y  +524.345, Z    +0.000, E1   -54.115, E3 +290668.641}
SPL {X  -165.650, Y  +531.171, Z    +0.000, E1   -54.075, E3 +290679.079}
SPL {X  -165.650, Y  +538.771, Z    +0.000, E1   -53.840, E3 +290691.820}
SPL {X  -165.650, Y  +548.103, Z    +0.000, E1   -53.944, E3 +290705.166}
SPL {X  -165.650, Y  +558.071, Z    +0.000, E1   -53.870, E3 +290720.507}
SPL {X  -165.650, Y  +568.053, Z    +0.000, E1   -54.124, E3 +290733.685}
SPL {X  -165.650, Y  +577.021, Z    +0.000, E1   -53.813, E3 +290749.183}
SPL {X  -165.650, Y  +587.996, Z    +0.000, E1   -53.969, E3 +290764.421}
SPL {X  -165.650, Y  +595.185, Z    +0.000, E1   -53.962, E3 +290775.130}
SPL {X  -165.650, Y  +602.138, Z    +0.000, E1   -53.941, E3 +290785.625}
SPL {X  -165.650, Y  +610.307, Z    +0.000, E1   -53.995, E3 +290797.472}
SPL {X  -165.650, Y  +617.878, Z    +0.000, E1   -53.838, E3 +290809.729}
SPL {X  -165.650, Y  +626.374, Z    +0.000, E1   -54.092, E3 +290820.744}
SPL {X  -165.650, Y  +632.964, Z    +0.000, E1   -53.887, E3 +290831.872}
SPL {X  -165.650, Y  +640.262, Z    +0.000, E1   -53.965, E3 +290842.187}
SPL {X  -165.650, Y  +647.911, Z    +0.000, E1   -53.930, E3 +290853.941}
SPL {X  -165.650, Y  +656.836, Z    +0.000, E1   -54.184, E3 +290865.473}
SPL {X  -165.650, Y  +659.513, Z    +0.000, E1   -53.578, E3 +290873.203}
SPL {X  -165.650, Y  +667.820, Z    +0.000, E1   -53.975, E3 +290883.268}
SPL {X  -165.623, Y  +678.503, Z    +0.000, E1   -53.932, E3 +290899.619}
SPL {X  -165.171, Y  +688.090, Z    +0.000, E1   -54.025, E3 +290913.067}
SPL {X  -164.558, Y  +694.489, Z    +0.000, E1   -53.745, E3 +290924.416}
SPL {X  -163.580, Y  +701.606, Z    +0.000, E1   -53.591, E3 +290935.849}
SPL {X  -162.702, Y  +706.614, Z    +0.000, E1   -53.230, E3 +290945.516}
SPL {X  -160.941, Y  +714.715, Z    +0.000, E1   -53.321, E3 +290957.136}
SPL {X  -159.638, Y  +719.723, Z    +0.000, E1   -52.685, E3 +290968.138}
SPL {X  -157.868, Y  +725.674, Z    +0.000, E1   -52.862, E3 +290975.995}
SPL {X  -156.314, Y  +730.327, Z    +0.000, E1   -52.199, E3 +290986.676}
SPL {X  -153.975, Y  +736.588, Z    +0.000, E1   -51.877, E3 +290997.707}
SPL {X  -151.949, Y  +741.465, Z    +0.000, E1   -51.645, E3 +291006.112}
SPL {X  -149.075, Y  +747.727, Z    +0.000, E1   -52.134, E3 +291012.827}
SPL {X  -137.775, Y  +767.467, Z    +0.000, E1   -56.912, E3 +291015.490}
SPL {X  -128.847, Y  +779.607, Z    +0.000, E1   -49.118, E3 +291090.506}
SPL {X   -94.133, Y  +811.804, Z    +0.000, E1   -53.019, E3 +291145.141}
ENDSPLINE

SPLINE
SPL {X  -123.886, Y  +785.464, Z    +0.000, E1   -49.465, E3 +291230.167}
SPL {X  -152.385, Y  +740.452, Z    +0.000, E1   -34.821, E3 +291211.144}
SPL {X  -162.077, Y  +709.719, Z    +0.000, E1   -21.590, E3 +291212.990}
SPL {X  -164.499, Y  +694.994, Z    +0.000, E1   -13.860, E3 +291213.775}
SPL {X  -165.382, Y  +684.927, Z    +0.000, E1    -7.984, E3 +291211.952}
SPL {X  -165.645, Y  +676.778, Z    +0.000, E1    -2.777, E3 +291211.675}
SPL {X  -165.650, Y  +672.938, Z    +0.000, E1    +0.157, E3 +291210.434}
SPL {X  -165.650, Y  +669.402, Z    +0.000, E1    +3.448, E3 +291209.825}
SPL {X  -165.650, Y  +663.061, Z    +0.000, E1   +11.076, E3 +291208.819}
SPL {X  -165.650, Y  +654.085, Z    +0.000, E1   +23.232, E3 +291207.926}
SPL {X  -165.650, Y  +639.700, Z    +0.000, E1   +43.326, E3 +291202.054}
SPL {X  -165.650, Y  +605.320, Z    +0.000, E1   +76.562, E3 +291181.463}
SPL {X  -165.650, Y  +596.505, Z    +0.000, E1   +55.802, E3 +291230.819}
SPL {X  -165.650, Y  +524.050, Z    +0.000, E1   +59.300, E3 +291294.978}
ENDSPLINE

SPLINE
SPL {X  -165.650, Y  +539.856, Z    +0.000, E1   +53.398, E3 +291310.626}
ENDSPLINE

SPLINE
SPL {X  -165.650, Y  +530.389, Z    +0.000, E1   +53.621, E3 +291323.631}
SPL {X  -165.650, Y  +521.849, Z    +0.000, E1   +53.452, E3 +291337.571}
SPL {X  -165.650, Y  +515.134, Z    +0.000, E1   +53.252, E3 +291348.922}
SPL {X  -165.650, Y  +505.685, Z    +0.000, E1   +53.701, E3 +291360.529}
SPL {X  -165.650, Y  +498.275, Z    +0.000, E1   +53.357, E3 +291373.837}
SPL {X  -165.650, Y  +491.031, Z    +0.000, E1   +53.348, E3 +291384.857}
SPL {X  -165.650, Y  +479.077, Z    +0.000, E1   +55.039, E3 +291391.980}
SPL {X  -165.650, Y  +450.615, Z    +0.000, E1   +59.721, E3 +291398.486}
SPL {X  -165.650, Y  +449.326, Z    +0.000, E1   +58.606, E3 +291407.535}
SPL {X  -165.650, Y  +442.154, Z    +0.000, E1   +58.369, E3 +291418.159}
SPL {X  -165.650, Y  +437.405, Z    +0.000, E1   +57.663, E3 +291428.769}
SPL {X  -165.650, Y  +432.227, Z    +0.000, E1   +57.103, E3 +291439.256}
SPL {X  -165.650, Y  +428.683, Z    +0.000, E1   +56.222, E3 +291449.611}
SPL {X  -165.650, Y  +424.202, Z    +0.000, E1   +55.382, E3 +291461.300}
SPL {X  -165.650, Y  +420.516, Z    +0.000, E1   +54.144, E3 +291474.305}
SPL {X  -165.650, Y  +412.197, Z    +0.000, E1   +54.057, E3 +291487.226}
SPL {X  -165.650, Y  +405.379, Z    +0.000, E1   +53.922, E3 +291498.093}
SPL {X  -165.650, Y  +400.791, Z    +0.000, E1   +53.827, E3 +291505.507}
SPL {X  -165.650, Y  +391.401, Z    +0.000, E1   +53.934, E3 +291519.106}
SPL {X  -165.650, Y  +378.987, Z    +0.000, E1   +53.974, E3 +291537.303}
SPL {X  -165.408, Y  +369.556, Z    +0.000, E1   +53.942, E3 +291551.394}
SPL {X  -164.927, Y  +363.041, Z    +0.000, E1   +53.687, E3 +291562.690}
SPL {X  -163.980, Y  +355.035, Z    +0.000, E1   +53.657, E3 +291574.886}
SPL {X  -162.665, Y  +347.197, Z    +0.000, E1   +53.396, E3 +291588.149}
SPL {X  -161.218, Y  +340.437, Z    +0.000, E1   +53.207, E3 +291599.248}
SPL {X  -159.523, Y  +333.864, Z    +0.000, E1   +52.908, E3 +291610.870}
SPL {X  -157.624, Y  +327.563, Z    +0.000, E1   +52.705, E3 +291621.280}
SPL {X  -156.289, Y  +323.602, Z    +0.000, E1   +52.159, E3 +291630.168}
SPL {X  -153.877, Y  +317.168, Z    +0.000, E1   +51.945, E3 +291641.030}
SPL {X  -151.035, Y  +310.467, Z    +0.000, E1   +51.312, E3 +291654.275}
SPL {X  -139.567, Y  +289.276, Z    +0.000, E1   +56.334, E3 +291658.363}
SPL {X  -117.053, Y  +261.289, Z    +0.000, E1   +49.815, E3 +291771.897}
ENDSPLINE

SPLINE
SPL {X  -148.836, Y  +305.783, Z    +0.000, E1   +38.029, E3 +291863.375}
SPL {X  -161.816, Y  +343.065, Z    +0.000, E1   +22.147, E3 +291854.025}
SPL {X  -164.614, Y  +360.007, Z    +0.000, E1   +13.213, E3 +291849.811}
SPL {X  -165.520, Y  +371.933, Z    +0.000, E1    +6.276, E3 +291852.565}
SPL {X  -165.650, Y  +378.704, Z    +0.000, E1    +1.700, E3 +291851.435}
SPL {X  -165.650, Y  +382.197, Z    +0.000, E1    -1.038, E3 +291850.508}
SPL {X  -165.650, Y  +386.782, Z    +0.000, E1    -5.783, E3 +291849.986}
SPL {X  -165.650, Y  +392.406, Z    +0.000, E1   -13.042, E3 +291847.883}
SPL {X  -165.650, Y  +398.038, Z    +0.000, E1   -20.113, E3 +291849.450}
SPL {X  -165.650, Y  +403.005, Z    +0.000, E1   -26.762, E3 +291848.632}
SPL {X  -165.650, Y  +415.469, Z    +0.000, E1   -43.461, E3 +291843.455}
SPL {X  -165.650, Y  +460.095, Z    +0.000, E1   -60.221, E3 +291861.717}
SPL {X  -165.650, Y  +535.749, Z    +0.000, E1   -60.559, E3 +291932.560}
ENDSPLINE

SPLINE
SPL {X  -165.650, Y  +516.750, Z    +0.000, E1   -54.244, E3 +291948.411}
ENDSPLINE

SPLINE
SPL {X  -165.650, Y  +524.345, Z    +0.000, E1   -54.115, E3 +291960.308}
SPL {X  -165.650, Y  +531.171, Z    +0.000, E1   -54.075, E3 +291970.746}
SPL {X  -165.650, Y  +538.771, Z    +0.000, E1   -53.840, E3 +291983.486}
SPL {X  -165.650, Y  +545.884, Z    +0.000, E1   -53.883, E3 +291993.791}
SPL {X  -165.650, Y  +553.081, Z    +0.000, E1   -53.834, E3 +292004.924}
SPL {X  -165.650, Y  +560.989, Z    +0.000, E1   -53.974, E3 +292015.761}
SPL {X  -165.650, Y  +568.053, Z    +0.000, E1   -54.124, E3 +292025.351}
SPL {X  -165.650, Y  +577.021, Z    +0.000, E1   -53.813, E3 +292040.850}
SPL {X  -165.650, Y  +587.996, Z    +0.000, E1   -53.969, E3 +292056.088}
SPL {X  -165.650, Y  +595.185, Z    +0.000, E1   -53.962, E3 +292066.797}
SPL {X  -165.650, Y  +602.138, Z    +0.000, E1   -53.941, E3 +292077.291}
SPL {X  -165.650, Y  +610.307, Z    +0.000, E1   -53.995, E3 +292089.139}
SPL {X  -165.650, Y  +617.878, Z    +0.000, E1   -53.838, E3 +292101.396}
SPL {X  -165.650, Y  +626.374, Z    +0.000, E1   -54.092, E3 +292112.411}
SPL {X  -165.650, Y  +632.964, Z    +0.000, E1   -53.887, E3 +292123.539}
SPL {X  -165.650, Y  +643.032, Z    +0.000, E1   -53.946, E3 +292138.283}
SPL {X  -165.650, Y  +654.069, Z    +0.000, E1   -54.108, E3 +292153.643}
SPL {X  -165.650, Y  +659.513, Z    +0.000, E1   -53.578, E3 +292164.869}
SPL {X  -165.650, Y  +667.820, Z    +0.000, E1   -53.975, E3 +292174.934}
SPL {X  -165.650, Y  +674.957, Z    +0.000, E1   -53.977, E3 +292185.447}
SPL {X  -165.574, Y  +680.515, Z    +0.000, E1   -53.820, E3 +292194.773}
SPL {X  -165.171, Y  +688.090, Z    +0.000, E1   -54.025, E3 +292204.734}
SPL {X  -164.558, Y  +694.489, Z    +0.000, E1   -53.745, E3 +292216.083}
SPL {X  -163.580, Y  +701.606, Z    +0.000, E1   -53.591, E3 +292227.516}
SPL {X  -162.702, Y  +706.614, Z    +0.000, E1   -53.230, E3 +292237.183}
SPL {X  -160.941, Y  +714.715, Z    +0.000, E1   -53.321, E3 +292248.802}
SPL {X  -159.638, Y  +719.723, Z    +0.000, E1   -52.685, E3 +292259.805}
SPL {X  -157.868, Y  +725.674, Z    +0.000, E1   -52.862, E3 +292267.662}
SPL {X  -156.314, Y  +730.327, Z    +0.000, E1   -52.199, E3 +292278.343}
SPL {X  -153.975, Y  +736.588, Z    +0.000, E1   -51.877, E3 +292289.373}
SPL {X  -151.949, Y  +741.465, Z    +0.000, E1   -51.645, E3 +292297.779}
SPL {X  -149.075, Y  +747.727, Z    +0.000, E1   -52.134, E3 +292304.493}
SPL {X  -137.775, Y  +767.467, Z    +0.000, E1   -56.912, E3 +292307.157}
SPL {X  -128.847, Y  +779.607, Z    +0.000, E1   -49.118, E3 +292382.173}
SPL {X   -94.133, Y  +811.804, Z    +0.000, E1   -53.019, E3 +292436.807}
ENDSPLINE

SPLINE
SPL {X  -134.098, Y  +772.750, Z    +0.000, E1   -45.587, E3 +292512.102}
SPL {X  -155.319, Y  +733.085, Z    +0.000, E1   -31.947, E3 +292502.979}
SPL {X  -162.077, Y  +709.719, Z    +0.000, E1   -21.590, E3 +292504.657}
SPL {X  -164.499, Y  +694.994, Z    +0.000, E1   -13.860, E3 +292505.442}
SPL {X  -165.382, Y  +684.927, Z    +0.000, E1    -7.984, E3 +292503.619}
SPL {X  -165.645, Y  +676.778, Z    +0.000, E1    -2.777, E3 +292503.341}
SPL {X  -165.650, Y  +672.041, Z    +0.000, E1    +0.844, E3 +292502.033}
SPL {X  -165.650, Y  +667.328, Z    +0.000, E1    +5.806, E3 +292501.410}
SPL {X  -165.650, Y  +661.774, Z    +0.000, E1   +13.006, E3 +292499.734}
SPL {X  -165.650, Y  +656.573, Z    +0.000, E1   +19.875, E3 +292500.292}
SPL {X  -165.650, Y  +650.769, Z    +0.000, E1   +28.083, E3 +292498.658}
SPL {X  -165.650, Y  +639.700, Z    +0.000, E1   +43.326, E3 +292493.720}
SPL {X  -165.650, Y  +605.320, Z    +0.000, E1   +76.562, E3 +292473.130}
SPL {X  -165.650, Y  +597.745, Z    +0.000, E1   +59.636, E3 +292511.131}
SPL {X  -165.650, Y  +596.360, Z    +0.000, E1   +54.978, E3 +292524.739}
SPL {X  -165.650, Y  +524.050, Z    +0.000, E1   +59.300, E3 +292586.645}
ENDSPLINE

SPLINE
SPL {X  -165.650, Y  +539.856, Z    +0.000, E1   +53.398, E3 +292602.292}
ENDSPLINE

SPLINE
SPL {X  -165.650, Y  +530.389, Z    +0.000, E1   +53.621, E3 +292615.298}
SPL {X  -165.650, Y  +521.849, Z    +0.000, E1   +53.452, E3 +292629.237}
SPL {X  -165.650, Y  +515.134, Z    +0.000, E1   +53.252, E3 +292640.588}
SPL {X  -165.650, Y  +505.685, Z    +0.000, E1   +53.701, E3 +292652.196}
SPL {X  -165.650, Y  +498.275, Z    +0.000, E1   +53.357, E3 +292665.504}
SPL {X  -165.650, Y  +487.031, Z    +0.000, E1   +53.931, E3 +292678.912}
SPL {X  -165.650, Y  +450.615, Z    +0.000, E1   +59.721, E3 +292690.152}
SPL {X  -165.650, Y  +449.326, Z    +0.000, E1   +58.606, E3 +292699.202}
SPL {X  -165.650, Y  +442.154, Z    +0.000, E1   +58.369, E3 +292709.826}
SPL {X  -165.650, Y  +437.405, Z    +0.000, E1   +57.663, E3 +292720.435}
SPL {X  -165.650, Y  +432.227, Z    +0.000, E1   +57.103, E3 +292730.923}
SPL {X  -165.650, Y  +428.683, Z    +0.000, E1   +56.222, E3 +292741.277}
SPL {X  -165.650, Y  +424.202, Z    +0.000, E1   +55.382, E3 +292752.966}
SPL {X  -165.650, Y  +418.469, Z    +0.000, E1   +54.594, E3 +292766.074}
SPL {X  -165.650, Y  +413.857, Z    +0.000, E1   +53.683, E3 +292778.645}
SPL {X  -165.650, Y  +403.104, Z    +0.000, E1   +53.908, E3 +292793.382}
SPL {X  -165.650, Y  +393.046, Z    +0.000, E1   +53.951, E3 +292808.066}
SPL {X  -165.650, Y  +383.306, Z    +0.000, E1   +53.987, E3 +292822.343}
SPL {X  -165.640, Y  +376.676, Z    +0.000, E1   +53.760, E3 +292833.510}
SPL {X  -165.408, Y  +369.556, Z    +0.000, E1   +53.942, E3 +292843.061}
SPL {X  -164.927, Y  +363.041, Z    +0.000, E1   +53.687, E3 +292854.356}
SPL {X  -163.980, Y  +355.035, Z    +0.000, E1   +53.657, E3 +292866.553}
SPL {X  -162.665, Y  +347.197, Z    +0.000, E1   +53.396, E3 +292879.816}
SPL {X  -161.218, Y  +340.437, Z    +0.000, E1   +53.207, E3 +292890.915}
SPL {X  -159.523, Y  +333.864, Z    +0.000, E1   +52.908, E3 +292902.537}
SPL {X  -157.624, Y  +327.563, Z    +0.000, E1   +52.705, E3 +292912.946}
SPL {X  -155.665, Y  +321.859, Z    +0.000, E1   +52.064, E3 +292925.119}
SPL {X  -152.682, Y  +314.249, Z    +0.000, E1   +51.841, E3 +292937.567}
SPL {X  -150.607, Y  +309.525, Z    +0.000, E1   +51.147, E3 +292948.052}
SPL {X  -142.104, Y  +293.374, Z    +0.000, E1   +55.775, E3 +292947.784}
SPL {X  -134.755, Y  +282.163, Z    +0.000, E1   +57.236, E3 +292954.052}
SPL {X  -117.053, Y  +261.289, Z    +0.000, E1   +49.815, E3 +293063.564}
ENDSPLINE

SPLINE
SPL {X  -148.836, Y  +305.783, Z    +0.000, E1   +38.029, E3 +293155.041}
SPL {X  -161.816, Y  +343.065, Z    +0.000, E1   +22.147, E3 +293145.691}
SPL {X  -164.614, Y  +360.007, Z    +0.000, E1   +13.213, E3 +293141.478}
SPL {X  -165.520, Y  +371.933, Z    +0.000, E1    +6.276, E3 +293144.232}
SPL {X  -165.650, Y  +378.704, Z    +0.000, E1    +1.700, E3 +293143.101}
SPL {X  -165.650, Y  +382.197, Z    +0.000, E1    -1.038, E3 +293142.175}
SPL {X  -165.650, Y  +386.782, Z    +0.000, E1    -5.783, E3 +293141.652}
SPL {X  -165.650, Y  +392.406, Z    +0.000, E1   -13.042, E3 +293139.550}
SPL {X  -165.650, Y  +398.038, Z    +0.000, E1   -20.113, E3 +293141.117}
SPL {X  -165.650, Y  +403.005, Z    +0.000, E1   -26.762, E3 +293140.299}
SPL {X  -165.650, Y  +415.469, Z    +0.000, E1   -43.461, E3 +293135.122}
SPL {X  -165.650, Y  +460.095, Z    +0.000, E1   -60.221, E3 +293153.383}
SPL {X  -165.650, Y  +537.366, Z    +0.000, E1   -61.810, E3 +293217.960}
ENDSPLINE

SPLINE
SPL {X  -165.650, Y  +520.647, Z    +0.000, E1   -55.836, E3 +293235.652}
ENDSPLINE

SPLINE
SPL {X  -165.650, Y  +521.328, Z    +0.000, E1   -53.870, E3 +293249.068}
SPL {X  -165.650, Y  +531.171, Z    +0.000, E1   -54.075, E3 +293262.413}
SPL {X  -165.650, Y  +538.771, Z    +0.000, E1   -53.840, E3 +293275.153}
SPL {X  -165.650, Y  +548.103, Z    +0.000, E1   -53.944, E3 +293288.500}
SPL {X  -165.650, Y  +558.071, Z    +0.000, E1   -53.870, E3 +293303.840}
SPL {X  -165.650, Y  +568.053, Z    +0.000, E1   -54.124, E3 +293317.018}
SPL {X  -165.650, Y  +574.396, Z    +0.000, E1   -53.807, E3 +293328.410}
SPL {X  -165.650, Y  +579.991, Z    +0.000, E1   -53.716, E3 +293337.319}
SPL {X  -165.650, Y  +587.996, Z    +0.000, E1   -53.969, E3 +293347.754}
SPL {X  -165.650, Y  +595.185, Z    +0.000, E1   -53.962, E3 +293358.464}
SPL {X  -165.650, Y  +602.138, Z    +0.000, E1   -53.941, E3 +293368.958}
SPL {X  -165.650, Y  +610.307, Z    +0.000, E1   -53.995, E3 +293380.806}
SPL {X  -165.650, Y  +617.878, Z    +0.000, E1   -53.838, E3 +293393.062}
SPL {X  -165.650, Y  +626.374, Z    +0.000, E1   -54.092, E3 +293404.078}
SPL {X  -165.650, Y  +632.964, Z    +0.000, E1   -53.887, E3 +293415.205}
SPL {X  -165.650, Y  +640.262, Z    +0.000, E1   -53.965, E3 +293425.520}
SPL {X  -165.650, Y  +647.911, Z    +0.000, E1   -53.930, E3 +293437.274}
SPL {X  -165.650, Y  +656.836, Z    +0.000, E1   -54.184, E3 +293448.806}
SPL {X  -165.650, Y  +659.513, Z    +0.000, E1   -53.578, E3 +293456.536}
SPL {X  -165.650, Y  +667.820, Z    +0.000, E1   -53.975, E3 +293466.601}
SPL {X  -165.623, Y  +678.503, Z    +0.000, E1   -53.932, E3 +293482.953}
SPL {X  -165.027, Y  +689.850, Z    +0.000, E1   -53.862, E3 +293500.216}
SPL {X  -163.840, Y  +699.919, Z    +0.000, E1   -53.732, E3 +293515.998}
SPL {X  -162.702, Y  +706.614, Z    +0.000, E1   -53.230, E3 +293528.849}
SPL {X  -161.265, Y  +713.361, Z    +0.000, E1   -53.436, E3 +293537.658}
SPL {X  -159.936, Y  +718.632, Z    +0.000, E1   -52.857, E3 +293548.987}
SPL {X  -157.868, Y  +725.674, Z    +0.000, E1   -52.862, E3 +293559.328}
SPL {X  -156.314, Y  +730.327, Z    +0.000, E1   -52.199, E3 +293570.010}
SPL {X  -153.975, Y  +736.588, Z    +0.000, E1   -51.877, E3 +293581.040}
SPL {X  -151.949, Y  +741.465, Z    +0.000, E1   -51.645, E3 +293589.445}
SPL {X  -149.075, Y  +747.727, Z    +0.000, E1   -52.134, E3 +293596.160}
SPL {X  -137.775, Y  +767.467, Z    +0.000, E1   -56.912, E3 +293598.823}
SPL {X  -128.847, Y  +779.607, Z    +0.000, E1   -49.118, E3 +293673.840}
SPL {X   -94.133, Y  +811.804, Z    +0.000, E1   -53.019, E3 +293728.474}
ENDSPLINE

SPLINE
SPL {X  -134.098, Y  +772.750, Z    +0.000, E1   -45.587, E3 +293803.768}
SPL {X  -155.319, Y  +733.085, Z    +0.000, E1   -31.947, E3 +293794.646}
SPL {X  -162.077, Y  +709.719, Z    +0.000, E1   -21.590, E3 +293796.324}
SPL {X  -164.499, Y  +694.994, Z    +0.000, E1   -13.860, E3 +293797.108}
SPL {X  -165.513, Y  +682.236, Z    +0.000, E1    -6.385, E3 +293795.444}
SPL {X  -165.650, Y  +675.776, Z    +0.000, E1    -2.014, E3 +293794.752}
SPL {X  -165.650, Y  +672.938, Z    +0.000, E1    +0.157, E3 +293793.767}
SPL {X  -165.650, Y  +669.402, Z    +0.000, E1    +3.448, E3 +293793.158}
SPL {X  -165.650, Y  +663.061, Z    +0.000, E1   +11.076, E3 +293792.152}
SPL {X  -165.650, Y  +656.573, Z    +0.000, E1   +19.875, E3 +293791.959}
SPL {X  -165.650, Y  +647.335, Z    +0.000, E1   +32.835, E3 +293788.881}
SPL {X  -165.650, Y  +637.438, Z    +0.000, E1   +46.409, E3 +293784.241}
SPL {X  -165.650, Y  +605.320, Z    +0.000, E1   +76.562, E3 +293764.796}
SPL {X  -165.650, Y  +596.505, Z    +0.000, E1   +55.802, E3 +293814.152}
SPL {X  -165.650, Y  +524.050, Z    +0.000, E1   +59.300, E3 +293878.312}
ENDSPLINE

SPLINE
SPL {X  -165.650, Y  +539.856, Z    +0.000, E1   +53.398, E3 +293893.959}
ENDSPLINE

SPLINE
SPL {X  -165.650, Y  +532.042, Z    +0.000, E1   +53.611, E3 +293904.430}
SPL {X  -165.650, Y  +526.147, Z    +0.000, E1   +53.495, E3 +293914.069}
SPL {X  -165.650, Y  +520.102, Z    +0.000, E1   +53.446, E3 +293923.495}
SPL {X  -165.650, Y  +512.447, Z    +0.000, E1   +53.456, E3 +293935.163}
SPL {X  -165.650, Y  +503.994, Z    +0.000, E1   +53.652, E3 +293946.602}
SPL {X  -165.650, Y  +498.275, Z    +0.000, E1   +53.357, E3 +293957.170}
SPL {X  -165.650, Y  +487.031, Z    +0.000, E1   +53.931, E3 +293970.579}
SPL {X  -165.650, Y  +450.615, Z    +0.000, E1   +59.721, E3 +293981.819}
SPL {X  -165.650, Y  +449.326, Z    +0.000, E1   +58.606, E3 +293990.868}
SPL {X  -165.650, Y  +442.154, Z    +0.000, E1   +58.369, E3 +294001.492}
SPL {X  -165.650, Y  +437.405, Z    +0.000, E1   +57.663, E3 +294012.102}
SPL {X  -165.650, Y  +432.227, Z    +0.000, E1   +57.103, E3 +294022.590}
SPL {X  -165.650, Y  +428.683, Z    +0.000, E1   +56.222, E3 +294032.944}
SPL {X  -165.650, Y  +424.202, Z    +0.000, E1   +55.382, E3 +294044.633}
SPL {X  -165.650, Y  +418.756, Z    +0.000, E1   +54.154, E3 +294060.312}
SPL {X  -165.650, Y  +410.508, Z    +0.000, E1   +54.007, E3 +294073.267}
SPL {X  -165.650, Y  +403.104, Z    +0.000, E1   +53.908, E3 +294085.049}
SPL {X  -165.650, Y  +393.046, Z    +0.000, E1   +53.951, E3 +294099.732}
SPL {X  -165.650, Y  +383.306, Z    +0.000, E1   +53.987, E3 +294114.010}
SPL {X  -165.600, Y  +374.450, Z    +0.000, E1   +53.824, E3 +294128.211}
SPL {X  -165.050, Y  +364.408, Z    +0.000, E1   +53.830, E3 +294143.270}
SPL {X  -164.096, Y  +355.862, Z    +0.000, E1   +53.838, E3 +294155.753}
SPL {X  -163.142, Y  +349.785, Z    +0.000, E1   +53.493, E3 +294166.969}
SPL {X  -161.604, Y  +342.113, Z    +0.000, E1   +53.155, E3 +294180.463}
SPL {X  -160.424, Y  +337.221, Z    +0.000, E1   +52.694, E3 +294190.303}
SPL {X  -158.192, Y  +329.354, Z    +0.000, E1   +52.890, E3 +294201.135}
SPL {X  -156.289, Y  +323.602, Z    +0.000, E1   +52.159, E3 +294213.502}
SPL {X  -154.898, Y  +319.792, Z    +0.000, E1   +51.850, E3 +294220.837}
SPL {X  -152.682, Y  +314.249, Z    +0.000, E1   +51.841, E3 +294229.234}
SPL {X  -150.607, Y  +309.525, Z    +0.000, E1   +51.147, E3 +294239.719}
SPL {X  -142.104, Y  +293.374, Z    +0.000, E1   +55.775, E3 +294239.450}
SPL {X  -134.755, Y  +282.163, Z    +0.000, E1   +57.236, E3 +294245.719}
SPL {X  -117.053, Y  +261.289, Z    +0.000, E1   +49.815, E3 +294355.230}
ENDSPLINE

SPLINE
SPL {X  -148.836, Y  +305.783, Z    +0.000, E1   +38.029, E3 +294446.708}
SPL {X  -161.816, Y  +343.065, Z    +0.000, E1   +22.147, E3 +294437.358}
SPL {X  -165.007, Y  +363.921, Z    +0.000, E1   +11.079, E3 +294435.347}
SPL {X  -165.587, Y  +373.939, Z    +0.000, E1    +4.928, E3 +294435.187}
SPL {X  -165.650, Y  +380.164, Z    +0.000, E1    +0.707, E3 +294434.368}
SPL {X  -165.650, Y  +384.850, Z    +0.000, E1    -3.598, E3 +294433.475}
SPL {X  -165.650, Y  +391.255, Z    +0.000, E1   -11.346, E3 +294431.817}
SPL {X  -165.650, Y  +398.038, Z    +0.000, E1   -20.113, E3 +294432.784}
SPL {X  -165.650, Y  +403.005, Z    +0.000, E1   -26.762, E3 +294431.966}
SPL {X  -165.650, Y  +415.469, Z    +0.000, E1   -43.461, E3 +294426.789}
SPL {X  -165.650, Y  +460.095, Z    +0.000, E1   -60.221, E3 +294445.050}
SPL {X  -165.650, Y  +535.749, Z    +0.000, E1   -60.559, E3 +294515.894}
ENDSPLINE

SPLINE
SPL {X  -165.650, Y  +516.866, Z    +0.000, E1   -54.768, E3 +294528.444}
ENDSPLINE

SPLINE
SPL {X  -165.650, Y  +521.328, Z    +0.000, E1   -53.870, E3 +294540.735}
SPL {X  -165.650, Y  +531.171, Z    +0.000, E1   -54.075, E3 +294554.079}
SPL {X  -165.650, Y  +538.771, Z    +0.000, E1   -53.840, E3 +294566.820}
SPL {X  -165.650, Y  +545.884, Z    +0.000, E1   -53.883, E3 +294577.124}
SPL {X  -165.650, Y  +553.081, Z    +0.000, E1   -53.834, E3 +294588.257}
SPL {X  -165.650, Y  +560.989, Z    +0.000, E1   -53.974, E3 +294599.094}
SPL {X  -165.650, Y  +568.053, Z    +0.000, E1   -54.124, E3 +294608.685}
SPL {X  -165.650, Y  +577.021, Z    +0.000, E1   -53.813, E3 +294624.183}
SPL {X  -165.650, Y  +587.996, Z    +0.000, E1   -53.969, E3 +294639.421}
SPL {X  -165.650, Y  +595.185, Z    +0.000, E1   -53.962, E3 +294650.130}
SPL {X  -165.650, Y  +602.138, Z    +0.000, E1   -53.941, E3 +294660.625}
SPL {X  -165.650, Y  +610.307, Z    +0.000, E1   -53.995, E3 +294672.472}
SPL {X  -165.650, Y  +617.878, Z    +0.000, E1   -53.838, E3 +294684.729}
SPL {X  -165.650, Y  +626.374, Z    +0.000, E1   -54.092, E3 +294695.744}
SPL {X  -165.650, Y  +632.964, Z    +0.000, E1   -53.887, E3 +294706.872}
SPL {X  -165.650, Y  +643.032, Z    +0.000, E1   -53.946, E3 +294721.616}
SPL {X  -165.650, Y  +654.069, Z    +0.000, E1   -54.108, E3 +294736.976}
SPL {X  -165.650, Y  +659.513, Z    +0.000, E1   -53.578, E3 +294748.203}
SPL {X  -165.650, Y  +667.820, Z    +0.000, E1   -53.975, E3 +294758.268}
SPL {X  -165.650, Y  +674.957, Z    +0.000, E1   -53.977, E3 +294768.780}
SPL {X  -165.574, Y  +680.515, Z    +0.000, E1   -53.820, E3 +294778.107}
SPL {X  -165.027, Y  +689.850, Z    +0.000, E1   -53.862, E3 +294791.883}
SPL {X  -163.840, Y  +699.919, Z    +0.000, E1   -53.732, E3 +294807.665}
SPL {X  -162.702, Y  +706.614, Z    +0.000, E1   -53.230, E3 +294820.516}
SPL {X  -160.941, Y  +714.715, Z    +0.000, E1   -53.321, E3 +294832.136}
SPL {X  -159.638, Y  +719.723, Z    +0.000, E1   -52.685, E3 +294843.138}
SPL {X  -157.868, Y  +725.674, Z    +0.000, E1   -52.862, E3 +294850.995}
SPL {X  -156.314, Y  +730.327, Z    +0.000, E1   -52.199, E3 +294861.676}
SPL {X  -153.975, Y  +736.588, Z    +0.000, E1   -51.877, E3 +294872.707}
SPL {X  -151.181, Y  +743.207, Z    +0.000, E1   -51.549, E3 +294884.327}
SPL {X  -146.528, Y  +752.763, Z    +0.000, E1   -53.481, E3 +294888.505}
SPL {X  -137.775, Y  +767.467, Z    +0.000, E1   -56.912, E3 +294890.490}
SPL {X  -128.847, Y  +779.607, Z    +0.000, E1   -49.118, E3 +294965.506}
SPL {X   -94.133, Y  +811.804, Z    +0.000, E1   -53.019, E3 +295020.141}
ENDSPLINE

SPLINE
SPL {X  -134.098, Y  +772.750, Z    +0.000, E1   -45.587, E3 +295095.435}
SPL {X  -155.319, Y  +733.085, Z    +0.000, E1   -31.947, E3 +295086.313}
SPL {X  -162.077, Y  +709.719, Z    +0.000, E1   -21.590, E3 +295087.990}
SPL {X  -164.499, Y  +694.994, Z    +0.000, E1   -13.860, E3 +295088.775}
SPL {X  -165.382, Y  +684.927, Z    +0.000, E1    -7.984, E3 +295086.952}
SPL {X  -165.645, Y  +676.778, Z    +0.000, E1    -2.777, E3 +295086.675}
SPL {X  -165.650, Y  +672.041, Z    +0.000, E1    +0.844, E3 +295085.366}
SPL {X  -165.650, Y  +667.328, Z    +0.000, E1    +5.806, E3 +295084.743}
SPL {X  -165.650, Y  +661.774, Z    +0.000, E1   +13.006, E3 +295083.067}
SPL {X  -165.650, Y  +656.573, Z    +0.000, E1   +19.875, E3 +295083.626}
SPL {X  -165.650, Y  +650.769, Z    +0.000, E1   +28.083, E3 +295081.992}
SPL {X  -165.650, Y  +639.700, Z    +0.000, E1   +43.326, E3 +295077.054}
SPL {X  -165.650, Y  +605.320, Z    +0.000, E1   +76.562, E3 +295056.463}
SPL {X  -165.650, Y  +597.745, Z    +0.000, E1   +59.636, E3 +295094.464}
SPL {X  -165.650, Y  +596.360, Z    +0.000, E1   +54.978, E3 +295108.072}
SPL {X  -165.650, Y  +524.050, Z    +0.000, E1   +59.300, E3 +295169.978}
ENDSPLINE

SPLINE
SPL {X  -165.650, Y  +539.856, Z    +0.000, E1   +53.398, E3 +295185.626}
ENDSPLINE

SPLINE
SPL {X  -165.650, Y  +530.389, Z    +0.000, E1   +53.621, E3 +295198.631}
SPL {X  -165.650, Y  +521.849, Z    +0.000, E1   +53.452, E3 +295212.571}
SPL {X  -165.650, Y  +515.134, Z    +0.000, E1   +53.252, E3 +295223.922}
SPL {X  -165.650, Y  +505.685, Z    +0.000, E1   +53.701, E3 +295235.529}
SPL {X  -165.650, Y  +498.275, Z    +0.000, E1   +53.357, E3 +295248.837}
SPL {X  -165.650, Y  +491.031, Z    +0.000, E1   +53.348, E3 +295259.857}
SPL {X  -165.650, Y  +479.077, Z    +0.000, E1   +55.039, E3 +295266.980}
SPL {X  -165.650, Y  +450.615, Z    +0.000, E1   +59.721, E3 +295273.486}
SPL {X  -165.650, Y  +449.326, Z    +0.000, E1   +58.606, E3 +295282.535}
SPL {X  -165.650, Y  +442.154, Z    +0.000, E1   +58.369, E3 +295293.159}
SPL {X  -165.650, Y  +437.405, Z    +0.000, E1   +57.663, E3 +295303.769}
SPL {X  -165.650, Y  +432.227, Z    +0.000, E1   +57.103, E3 +295314.256}
SPL {X  -165.650, Y  +428.683, Z    +0.000, E1   +56.222, E3 +295324.611}
SPL {X  -165.650, Y  +424.202, Z    +0.000, E1   +55.382, E3 +295336.300}
SPL {X  -165.650, Y  +418.756, Z    +0.000, E1   +54.154, E3 +295351.979}
SPL {X  -165.650, Y  +407.872, Z    +0.000, E1   +54.003, E3 +295369.064}
SPL {X  -165.650, Y  +400.791, Z    +0.000, E1   +53.827, E3 +295380.507}
SPL {X  -165.650, Y  +393.046, Z    +0.000, E1   +53.951, E3 +295391.399}
SPL {X  -165.650, Y  +383.306, Z    +0.000, E1   +53.987, E3 +295405.676}
SPL {X  -165.640, Y  +376.676, Z    +0.000, E1   +53.760, E3 +295416.843}
SPL {X  -165.408, Y  +369.556, Z    +0.000, E1   +53.942, E3 +295426.394}
SPL {X  -164.927, Y  +363.041, Z    +0.000, E1   +53.687, E3 +295437.690}
SPL {X  -164.096, Y  +355.862, Z    +0.000, E1   +53.838, E3 +295447.420}
SPL {X  -162.936, Y  +348.637, Z    +0.000, E1   +53.390, E3 +295461.136}
SPL {X  -161.218, Y  +340.437, Z    +0.000, E1   +53.207, E3 +295474.248}
SPL {X  -159.523, Y  +333.864, Z    +0.000, E1   +52.908, E3 +295485.870}
SPL {X  -157.624, Y  +327.563, Z    +0.000, E1   +52.705, E3 +295496.280}
SPL {X  -155.665, Y  +321.859, Z    +0.000, E1   +52.064, E3 +295508.453}
SPL {X  -152.682, Y  +314.249, Z    +0.000, E1   +51.841, E3 +295520.901}
SPL {X  -150.607, Y  +309.525, Z    +0.000, E1   +51.147, E3 +295531.385}
SPL {X  -142.104, Y  +293.374, Z    +0.000, E1   +55.775, E3 +295531.117}
SPL {X  -134.755, Y  +282.163, Z    +0.000, E1   +57.236, E3 +295537.385}
SPL {X  -117.053, Y  +261.289, Z    +0.000, E1   +49.815, E3 +295646.897}
ENDSPLINE

SPLINE
SPL {X  -148.836, Y  +305.783, Z    +0.000, E1   +38.029, E3 +295738.375}
SPL {X  -161.816, Y  +343.065, Z    +0.000, E1   +22.147, E3 +295729.025}
SPL {X  -164.614, Y  +360.007, Z    +0.000, E1   +13.213, E3 +295724.811}
SPL {X  -165.520, Y  +371.933, Z    +0.000, E1    +6.276, E3 +295727.565}
SPL {X  -165.650, Y  +378.704, Z    +0.000, E1    +1.700, E3 +295726.435}
SPL {X  -165.650, Y  +382.197, Z    +0.000, E1    -1.038, E3 +295725.508}
SPL {X  -165.650, Y  +386.782, Z    +0.000, E1    -5.783, E3 +295724.986}
SPL {X  -165.650, Y  +392.406, Z    +0.000, E1   -13.042, E3 +295722.883}
SPL {X  -165.650, Y  +398.038, Z    +0.000, E1   -20.113, E3 +295724.450}
SPL {X  -165.650, Y  +403.005, Z    +0.000, E1   -26.762, E3 +295723.632}
SPL {X  -165.650, Y  +415.469, Z    +0.000, E1   -43.461, E3 +295718.455}
SPL {X  -165.650, Y  +460.095, Z    +0.000, E1   -60.221, E3 +295736.717}
SPL {X  -165.650, Y  +535.749, Z    +0.000, E1   -60.559, E3 +295807.560}
ENDSPLINE

SPLINE
SPL {X  -165.650, Y  +516.750, Z    +0.000, E1   -54.244, E3 +295823.411}
ENDSPLINE

SPLINE
SPL {X  -165.650, Y  +524.345, Z    +0.000, E1   -54.115, E3 +295835.308}
SPL {X  -165.650, Y  +531.171, Z    +0.000, E1   -54.075, E3 +295845.746}
SPL {X  -165.650, Y  +538.771, Z    +0.000, E1   -53.840, E3 +295858.486}
SPL {X  -165.650, Y  +545.884, Z    +0.000, E1   -53.883, E3 +295868.791}
SPL {X  -165.650, Y  +553.081, Z    +0.000, E1   -53.834, E3 +295879.924}
SPL {X  -165.650, Y  +560.989, Z    +0.000, E1   -53.974, E3 +295890.761}
SPL {X  -165.650, Y  +568.053, Z    +0.000, E1   -54.124, E3 +295900.351}
SPL {X  -165.650, Y  +577.021, Z    +0.000, E1   -53.813, E3 +295915.850}
SPL {X  -165.650, Y  +587.996, Z    +0.000, E1   -53.969, E3 +295931.088}
SPL {X  -165.650, Y  +595.185, Z    +0.000, E1   -53.962, E3 +295941.797}
SPL {X  -165.650, Y  +602.138, Z    +0.000, E1   -53.941, E3 +295952.291}
SPL {X  -165.650, Y  +610.307, Z    +0.000, E1   -53.995, E3 +295964.139}
SPL {X  -165.650, Y  +617.878, Z    +0.000, E1   -53.838, E3 +295976.396}
SPL {X  -165.650, Y  +626.374, Z    +0.000, E1   -54.092, E3 +295987.411}
SPL {X  -165.650, Y  +632.964, Z    +0.000, E1   -53.887, E3 +295998.539}
SPL {X  -165.650, Y  +643.032, Z    +0.000, E1   -53.946, E3 +296013.283}
SPL {X  -165.650, Y  +654.069, Z    +0.000, E1   -54.108, E3 +296028.643}
SPL {X  -165.650, Y  +659.513, Z    +0.000, E1   -53.578, E3 +296039.869}
SPL {X  -165.650, Y  +667.820, Z    +0.000, E1   -53.975, E3 +296049.934}
SPL {X  -165.650, Y  +674.957, Z    +0.000, E1   -53.977, E3 +296060.447}
SPL {X  -165.574, Y  +680.515, Z    +0.000, E1   -53.820, E3 +296069.773}
SPL {X  -165.171, Y  +688.090, Z    +0.000, E1   -54.025, E3 +296079.734}
SPL {X  -164.558, Y  +694.489, Z    +0.000, E1   -53.745, E3 +296091.083}
SPL {X  -163.580, Y  +701.606, Z    +0.000, E1   -53.591, E3 +296102.516}
SPL {X  -162.702, Y  +706.614, Z    +0.000, E1   -53.230, E3 +296112.183}
SPL {X  -161.265, Y  +713.361, Z    +0.000, E1   -53.436, E3 +296120.991}
SPL {X  -159.936, Y  +718.632, Z    +0.000, E1   -52.857, E3 +296132.321}
SPL {X  -157.868, Y  +725.674, Z    +0.000, E1   -52.862, E3 +296142.662}
SPL {X  -156.314, Y  +730.327, Z    +0.000, E1   -52.199, E3 +296153.343}
SPL {X  -153.975, Y  +736.588, Z    +0.000, E1   -51.877, E3 +296164.373}
SPL {X  -151.181, Y  +743.207, Z    +0.000, E1   -51.549, E3 +296175.994}
SPL {X  -146.528, Y  +752.763, Z    +0.000, E1   -53.481, E3 +296180.171}
SPL {X  -137.775, Y  +767.467, Z    +0.000, E1   -56.912, E3 +296182.157}
SPL {X  -128.847, Y  +779.607, Z    +0.000, E1   -49.118, E3 +296257.173}
SPL {X   -94.133, Y  +811.804, Z    +0.000, E1   -53.019, E3 +296311.807}
ENDSPLINE

SPLINE
SPL {X  -123.886, Y  +785.464, Z    +0.000, E1   -49.465, E3 +296396.834}
SPL {X  -152.385, Y  +740.452, Z    +0.000, E1   -34.821, E3 +296377.811}
SPL {X  -162.077, Y  +709.719, Z    +0.000, E1   -21.590, E3 +296379.657}
SPL {X  -164.499, Y  +694.994, Z    +0.000, E1   -13.860, E3 +296380.442}
SPL {X  -165.513, Y  +682.236, Z    +0.000, E1    -6.385, E3 +296378.777}
SPL {X  -165.650, Y  +675.776, Z    +0.000, E1    -2.014, E3 +296378.085}
SPL {X  -165.650, Y  +672.041, Z    +0.000, E1    +0.844, E3 +296377.033}
SPL {X  -165.650, Y  +667.328, Z    +0.000, E1    +5.806, E3 +296376.410}
SPL {X  -165.650, Y  +661.774, Z    +0.000, E1   +13.006, E3 +296374.734}
SPL {X  -165.650, Y  +654.085, Z    +0.000, E1   +23.232, E3 +296374.593}
SPL {X  -165.650, Y  +639.700, Z    +0.000, E1   +43.326, E3 +296368.720}
SPL {X  -165.650, Y  +605.320, Z    +0.000, E1   +76.562, E3 +296348.130}
SPL {X  -165.650, Y  +597.745, Z    +0.000, E1   +59.636, E3 +296386.131}
SPL {X  -165.650, Y  +596.360, Z    +0.000, E1   +54.978, E3 +296399.739}
SPL {X  -165.650, Y  +524.050, Z    +0.000, E1   +59.300, E3 +296461.645}
ENDSPLINE

SPLINE
SPL {X  -165.650, Y  +539.856, Z    +0.000, E1   +53.398, E3 +296477.292}
ENDSPLINE

SPLINE
SPL {X  -165.650, Y  +530.389, Z    +0.000, E1   +53.621, E3 +296490.298}
SPL {X  -165.650, Y  +521.849, Z    +0.000, E1   +53.452, E3 +296504.237}
SPL {X  -165.650, Y  +515.134, Z    +0.000, E1   +53.252, E3 +296515.588}
SPL {X  -165.650, Y  +505.685, Z    +0.000, E1   +53.701, E3 +296527.196}
SPL {X  -165.650, Y  +498.275, Z    +0.000, E1   +53.357, E3 +296540.504}
SPL {X  -165.650, Y  +491.031, Z    +0.000, E1   +53.348, E3 +296551.524}
SPL {X  -165.650, Y  +479.077, Z    +0.000, E1   +55.039, E3 +296558.647}
SPL {X  -165.650, Y  +450.615, Z    +0.000, E1   +59.721, E3 +296565.152}
SPL {X  -165.650, Y  +449.326, Z    +0.000, E1   +58.606, E3 +296574.202}
SPL {X  -165.650, Y  +442.154, Z    +0.000, E1   +58.369, E3 +296584.826}
SPL {X  -165.650, Y  +437.405, Z    +0.000, E1   +57.663, E3 +296595.435}
SPL {X  -165.650, Y  +432.227, Z    +0.000, E1   +57.103, E3 +296605.923}
SPL {X  -165.650, Y  +428.683, Z    +0.000, E1   +56.222, E3 +296616.277}
SPL {X  -165.650, Y  +424.202, Z    +0.000, E1   +55.382, E3 +296627.966}
SPL {X  -165.650, Y  +418.756, Z    +0.000, E1   +54.154, E3 +296643.645}
SPL {X  -165.650, Y  +410.508, Z    +0.000, E1   +54.007, E3 +296656.601}
SPL {X  -165.650, Y  +403.104, Z    +0.000, E1   +53.908, E3 +296668.382}
SPL {X  -165.650, Y  +391.401, Z    +0.000, E1   +53.934, E3 +296685.773}
SPL {X  -165.650, Y  +378.987, Z    +0.000, E1   +53.974, E3 +296703.969}
SPL {X  -165.408, Y  +369.556, Z    +0.000, E1   +53.942, E3 +296718.061}
SPL {X  -164.927, Y  +363.041, Z    +0.000, E1   +53.687, E3 +296729.356}
SPL {X  -164.096, Y  +355.862, Z    +0.000, E1   +53.838, E3 +296739.087}
SPL {X  -163.142, Y  +349.785, Z    +0.000, E1   +53.493, E3 +296750.302}
SPL {X  -161.604, Y  +342.113, Z    +0.000, E1   +53.155, E3 +296763.797}
SPL {X  -160.424, Y  +337.221, Z    +0.000, E1   +52.694, E3 +296773.637}
SPL {X  -158.192, Y  +329.354, Z    +0.000, E1   +52.890, E3 +296784.468}
SPL {X  -156.289, Y  +323.602, Z    +0.000, E1   +52.159, E3 +296796.835}
SPL {X  -154.898, Y  +319.792, Z    +0.000, E1   +51.850, E3 +296804.170}
SPL {X  -152.682, Y  +314.249, Z    +0.000, E1   +51.841, E3 +296812.567}
SPL {X  -150.607, Y  +309.525, Z    +0.000, E1   +51.147, E3 +296823.052}
SPL {X  -139.567, Y  +289.276, Z    +0.000, E1   +56.334, E3 +296825.030}
SPL {X  -117.053, Y  +261.289, Z    +0.000, E1   +49.815, E3 +296938.564}
ENDSPLINE

SPLINE
SPL {X  -148.836, Y  +305.783, Z    +0.000, E1   +38.029, E3 +297030.041}
SPL {X  -161.816, Y  +343.065, Z    +0.000, E1   +22.147, E3 +297020.691}
SPL {X  -164.614, Y  +360.007, Z    +0.000, E1   +13.213, E3 +297016.478}
SPL {X  -165.520, Y  +371.933, Z    +0.000, E1    +6.276, E3 +297019.232}
SPL {X  -165.650, Y  +378.704, Z    +0.000, E1    +1.700, E3 +297018.101}
SPL {X  -165.650, Y  +382.197, Z    +0.000, E1    -1.038, E3 +297017.175}
SPL {X  -165.650, Y  +386.782, Z    +0.000, E1    -5.783, E3 +297016.652}
SPL {X  -165.650, Y  +392.406, Z    +0.000, E1   -13.042, E3 +297014.550}
SPL {X  -165.650, Y  +398.038, Z    +0.000, E1   -20.113, E3 +297016.117}
SPL {X  -165.650, Y  +403.005, Z    +0.000, E1   -26.762, E3 +297015.299}
SPL {X  -165.650, Y  +415.469, Z    +0.000, E1   -43.461, E3 +297010.122}
SPL {X  -165.650, Y  +460.095, Z    +0.000, E1   -60.221, E3 +297028.383}
SPL {X  -165.650, Y  +537.366, Z    +0.000, E1   -61.810, E3 +297092.960}
ENDSPLINE

SPLINE
SPL {X  -165.650, Y  +520.647, Z    +0.000, E1   -55.836, E3 +297110.652}
ENDSPLINE

SPLINE
SPL {X  -165.650, Y  +521.328, Z    +0.000, E1   -53.870, E3 +297124.068}
SPL {X  -165.650, Y  +531.171, Z    +0.000, E1   -54.075, E3 +297137.413}
SPL {X  -165.650, Y  +538.771, Z    +0.000, E1   -53.840, E3 +297150.153}
SPL {X  -165.650, Y  +548.103, Z    +0.000, E1   -53.944, E3 +297163.500}
SPL {X  -165.650, Y  +558.071, Z    +0.000, E1   -53.870, E3 +297178.840}
SPL {X  -165.650, Y  +568.053, Z    +0.000, E1   -54.124, E3 +297192.018}
SPL {X  -165.650, Y  +574.396, Z    +0.000, E1   -53.807, E3 +297203.410}
SPL {X  -165.650, Y  +579.991, Z    +0.000, E1   -53.716, E3 +297212.319}
SPL {X  -165.650, Y  +587.996, Z    +0.000, E1   -53.969, E3 +297222.754}
SPL {X  -165.650, Y  +595.185, Z    +0.000, E1   -53.962, E3 +297233.464}
SPL {X  -165.650, Y  +602.138, Z    +0.000, E1   -53.941, E3 +297243.958}
SPL {X  -165.650, Y  +610.307, Z    +0.000, E1   -53.995, E3 +297255.806}
SPL {X  -165.650, Y  +617.878, Z    +0.000, E1   -53.838, E3 +297268.062}
SPL {X  -165.650, Y  +626.374, Z    +0.000, E1   -54.092, E3 +297279.078}
SPL {X  -165.650, Y  +632.964, Z    +0.000, E1   -53.887, E3 +297290.205}
SPL {X  -165.650, Y  +640.262, Z    +0.000, E1   -53.965, E3 +297300.520}
SPL {X  -165.650, Y  +647.911, Z    +0.000, E1   -53.930, E3 +297312.274}
SPL {X  -165.650, Y  +656.836, Z    +0.000, E1   -54.184, E3 +297323.806}
SPL {X  -165.650, Y  +659.513, Z    +0.000, E1   -53.578, E3 +297331.536}
SPL {X  -165.650, Y  +667.820, Z    +0.000, E1   -53.975, E3 +297341.601}
SPL {X  -165.623, Y  +678.503, Z    +0.000, E1   -53.932, E3 +297357.953}
SPL {X  -165.027, Y  +689.850, Z    +0.000, E1   -53.862, E3 +297375.216}
SPL {X  -163.840, Y  +699.919, Z    +0.000, E1   -53.732, E3 +297390.998}
SPL {X  -162.702, Y  +706.614, Z    +0.000, E1   -53.230, E3 +297403.849}
SPL {X  -161.265, Y  +713.361, Z    +0.000, E1   -53.436, E3 +297412.658}
SPL {X  -159.936, Y  +718.632, Z    +0.000, E1   -52.857, E3 +297423.987}
SPL {X  -157.868, Y  +725.674, Z    +0.000, E1   -52.862, E3 +297434.328}
SPL {X  -156.314, Y  +730.327, Z    +0.000, E1   -52.199, E3 +297445.010}
SPL {X  -153.975, Y  +736.588, Z    +0.000, E1   -51.877, E3 +297456.040}
SPL {X  -151.949, Y  +741.465, Z    +0.000, E1   -51.645, E3 +297464.445}
SPL {X  -149.075, Y  +747.727, Z    +0.000, E1   -52.134, E3 +297471.160}
SPL {X  -137.775, Y  +767.467, Z    +0.000, E1   -56.912, E3 +297473.823}
SPL {X  -128.847, Y  +779.607, Z    +0.000, E1   -49.118, E3 +297548.840}
SPL {X   -94.133, Y  +811.804, Z    +0.000, E1   -53.019, E3 +297603.474}
ENDSPLINE

SPLINE
SPL {X  -134.098, Y  +772.750, Z    +0.000, E1   -45.587, E3 +297678.768}
SPL {X  -155.319, Y  +733.085, Z    +0.000, E1   -31.947, E3 +297669.646}
SPL {X  -162.077, Y  +709.719, Z    +0.000, E1   -21.590, E3 +297671.324}
SPL {X  -164.499, Y  +694.994, Z    +0.000, E1   -13.860, E3 +297672.108}
SPL {X  -165.513, Y  +682.236, Z    +0.000, E1    -6.385, E3 +297670.444}
SPL {X  -165.650, Y  +675.776, Z    +0.000, E1    -2.014, E3 +297669.752}
SPL {X  -165.650, Y  +672.938, Z    +0.000, E1    +0.157, E3 +297668.767}
SPL {X  -165.650, Y  +669.402, Z    +0.000, E1    +3.448, E3 +297668.158}
SPL {X  -165.650, Y  +663.061, Z    +0.000, E1   +11.076, E3 +297667.152}
SPL {X  -165.650, Y  +656.573, Z    +0.000, E1   +19.875, E3 +297666.959}
SPL {X  -165.650, Y  +650.769, Z    +0.000, E1   +28.083, E3 +297665.325}
SPL {X  -165.650, Y  +639.700, Z    +0.000, E1   +43.326, E3 +297660.387}
SPL {X  -165.650, Y  +605.320, Z    +0.000, E1   +76.562, E3 +297639.796}
SPL {X  -165.650, Y  +597.745, Z    +0.000, E1   +59.636, E3 +297677.798}
SPL {X  -165.650, Y  +596.360, Z    +0.000, E1   +54.978, E3 +297691.406}
SPL {X  -165.650, Y  +521.429, Z    +0.000, E1   +61.144, E3 +297744.637}
ENDSPLINE

SPLINE
SPL {X  -165.650, Y  +526.028, Z    +0.000, E1   +58.071, E3 +297758.411}
SPL {X  -165.650, Y  +539.856, Z    +0.000, E1   +53.398, E3 +297768.959}
ENDSPLINE

SPLINE
SPL {X  -165.650, Y  +532.042, Z    +0.000, E1   +53.611, E3 +297779.430}
SPL {X  -165.650, Y  +526.147, Z    +0.000, E1   +53.495, E3 +297789.069}
SPL {X  -165.650, Y  +517.365, Z    +0.000, E1   +53.387, E3 +297803.237}
SPL {X  -165.650, Y  +505.685, Z    +0.000, E1   +53.701, E3 +297818.863}
SPL {X  -165.650, Y  +498.275, Z    +0.000, E1   +53.357, E3 +297832.170}
SPL {X  -165.650, Y  +487.031, Z    +0.000, E1   +53.931, E3 +297845.579}
SPL {X  -165.650, Y  +450.615, Z    +0.000, E1   +59.721, E3 +297856.819}
SPL {X  -165.650, Y  +449.326, Z    +0.000, E1   +58.606, E3 +297865.868}
SPL {X  -165.650, Y  +442.154, Z    +0.000, E1   +58.369, E3 +297876.492}
SPL {X  -165.650, Y  +437.405, Z    +0.000, E1   +57.663, E3 +297887.102}
SPL {X  -165.650, Y  +432.227, Z    +0.000, E1   +57.103, E3 +297897.590}
SPL {X  -165.650, Y  +428.683, Z    +0.000, E1   +56.222, E3 +297907.944}
SPL {X  -165.650, Y  +424.202, Z    +0.000, E1   +55.382, E3 +297919.633}
SPL {X  -165.650, Y  +418.756, Z    +0.000, E1   +54.154, E3 +297935.312}
SPL {X  -165.650, Y  +410.508, Z    +0.000, E1   +54.007, E3 +297948.267}
SPL {X  -165.650, Y  +403.104, Z    +0.000, E1   +53.908, E3 +297960.049}
SPL {X  -165.650, Y  +393.046, Z    +0.000, E1   +53.951, E3 +297974.732}
SPL {X  -165.650, Y  +383.306, Z    +0.000, E1   +53.987, E3 +297989.010}
SPL {X  -165.640, Y  +376.676, Z    +0.000, E1   +53.760, E3 +298000.176}
SPL {X  -165.408, Y  +369.556, Z    +0.000, E1   +53.942, E3 +298009.727}
SPL {X  -164.927, Y  +363.041, Z    +0.000, E1   +53.687, E3 +298021.023}
SPL {X  -163.980, Y  +355.035, Z    +0.000, E1   +53.657, E3 +298033.219}
SPL {X  -162.665, Y  +347.197, Z    +0.000, E1   +53.396, E3 +298046.483}
SPL {X  -161.218, Y  +340.437, Z    +0.000, E1   +53.207, E3 +298057.581}
SPL {X  -159.523, Y  +333.864, Z    +0.000, E1   +52.908, E3 +298069.204}
SPL {X  -157.624, Y  +327.563, Z    +0.000, E1   +52.705, E3 +298079.613}
SPL {X  -156.289, Y  +323.602, Z    +0.000, E1   +52.159, E3 +298088.502}
SPL {X  -153.877, Y  +317.168, Z    +0.000, E1   +51.945, E3 +298099.363}
SPL {X  -151.035, Y  +310.467, Z    +0.000, E1   +51.312, E3 +298112.608}
SPL {X  -139.567, Y  +289.276, Z    +0.000, E1   +56.334, E3 +298116.697}
SPL {X  -117.053, Y  +261.289, Z    +0.000, E1   +49.815, E3 +298230.230}
ENDSPLINE

SPLINE
SPL {X  -148.836, Y  +305.783, Z    +0.000, E1   +38.029, E3 +298321.708}
SPL {X  -161.816, Y  +343.065, Z    +0.000, E1   +22.147, E3 +298312.358}
SPL {X  -164.614, Y  +360.007, Z    +0.000, E1   +13.213, E3 +298308.144}
SPL {X  -165.520, Y  +371.933, Z    +0.000, E1    +6.276, E3 +298310.899}
SPL {X  -165.650, Y  +378.704, Z    +0.000, E1    +1.700, E3 +298309.768}
SPL {X  -165.650, Y  +382.197, Z    +0.000, E1    -1.038, E3 +298308.841}
SPL {X  -165.650, Y  +386.782, Z    +0.000, E1    -5.783, E3 +298308.319}
SPL {X  -165.650, Y  +392.406, Z    +0.000, E1   -13.042, E3 +298306.216}
SPL {X  -165.650, Y  +400.489, Z    +0.000, E1   -23.243, E3 +298307.380}
SPL {X  -165.650, Y  +415.469, Z    +0.000, E1   -43.461, E3 +298301.789}
SPL {X  -165.650, Y  +460.095, Z    +0.000, E1   -60.221, E3 +298320.050}
SPL {X  -165.650, Y  +535.749, Z    +0.000, E1   -60.559, E3 +298390.894}
ENDSPLINE

SPLINE
SPL {X  -165.650, Y  +516.866, Z    +0.000, E1   -54.768, E3 +298403.444}
ENDSPLINE

SPLINE
SPL {X  -165.650, Y  +521.328, Z    +0.000, E1   -53.870, E3 +298415.735}
SPL {X  -165.650, Y  +531.171, Z    +0.000, E1   -54.075, E3 +298429.079}
SPL {X  -165.650, Y  +538.771, Z    +0.000, E1   -53.840, E3 +298441.820}
SPL {X  -165.650, Y  +548.103, Z    +0.000, E1   -53.944, E3 +298455.166}
SPL {X  -165.650, Y  +558.071, Z    +0.000, E1   -53.870, E3 +298470.507}
SPL {X  -165.650, Y  +568.053, Z    +0.000, E1   -54.124, E3 +298483.685}
SPL {X  -165.650, Y  +577.021, Z    +0.000, E1   -53.813, E3 +298499.183}
SPL {X  -165.650, Y  +587.996, Z    +0.000, E1   -53.969, E3 +298514.421}
SPL {X  -165.650, Y  +595.185, Z    +0.000, E1   -53.962, E3 +298525.130}
SPL {X  -165.650, Y  +602.138, Z    +0.000, E1   -53.941, E3 +298535.625}
SPL {X  -165.650, Y  +610.307, Z    +0.000, E1   -53.995, E3 +298547.472}
SPL {X  -165.650, Y  +617.878, Z    +0.000, E1   -53.838, E3 +298559.729}
SPL {X  -165.650, Y  +627.853, Z    +0.000, E1   -53.937, E3 +298574.083}
SPL {X  -165.650, Y  +638.510, Z    +0.000, E1   -54.057, E3 +298589.142}
SPL {X  -165.650, Y  +647.911, Z    +0.000, E1   -53.930, E3 +298603.941}
SPL {X  -165.650, Y  +658.189, Z    +0.000, E1   -53.932, E3 +298619.241}
SPL {X  -165.650, Y  +667.820, Z    +0.000, E1   -53.975, E3 +298633.268}
SPL {X  -165.623, Y  +678.503, Z    +0.000, E1   -53.932, E3 +298649.619}
SPL {X  -165.171, Y  +688.090, Z    +0.000, E1   -54.025, E3 +298663.067}
SPL {X  -164.558, Y  +694.489, Z    +0.000, E1   -53.745, E3 +298674.416}
SPL {X  -163.580, Y  +701.606, Z    +0.000, E1   -53.591, E3 +298685.849}
SPL {X  -162.702, Y  +706.614, Z    +0.000, E1   -53.230, E3 +298695.516}
SPL {X  -160.941, Y  +714.715, Z    +0.000, E1   -53.321, E3 +298707.136}
SPL {X  -159.638, Y  +719.723, Z    +0.000, E1   -52.685, E3 +298718.138}
SPL {X  -157.521, Y  +726.754, Z    +0.000, E1   -52.585, E3 +298729.334}
SPL {X  -155.632, Y  +732.234, Z    +0.000, E1   -52.209, E3 +298739.380}
SPL {X  -153.975, Y  +736.588, Z    +0.000, E1   -51.877, E3 +298747.707}
SPL {X  -151.949, Y  +741.465, Z    +0.000, E1   -51.645, E3 +298756.112}
SPL {X  -149.075, Y  +747.727, Z    +0.000, E1   -52.134, E3 +298762.827}
SPL {X  -137.775, Y  +767.467, Z    +0.000, E1   -56.912, E3 +298765.490}
SPL {X  -128.847, Y  +779.607, Z    +0.000, E1   -49.118, E3 +298840.506}
SPL {X   -94.133, Y  +811.804, Z    +0.000, E1   -53.019, E3 +298895.141}
ENDSPLINE

SPLINE
SPL {X  -134.098, Y  +772.750, Z    +0.000, E1   -45.587, E3 +298970.435}
SPL {X  -155.319, Y  +733.085, Z    +0.000, E1   -31.947, E3 +298961.313}
SPL {X  -162.077, Y  +709.719, Z    +0.000, E1   -21.590, E3 +298962.990}
SPL {X  -164.499, Y  +694.994, Z    +0.000, E1   -13.860, E3 +298963.775}
SPL {X  -165.382, Y  +684.927, Z    +0.000, E1    -7.984, E3 +298961.952}
SPL {X  -165.645, Y  +676.778, Z    +0.000, E1    -2.777, E3 +298961.675}
SPL {X  -165.650, Y  +672.041, Z    +0.000, E1    +0.844, E3 +298960.366}
SPL {X  -165.650, Y  +667.328, Z    +0.000, E1    +5.806, E3 +298959.743}
SPL {X  -165.650, Y  +661.774, Z    +0.000, E1   +13.006, E3 +298958.067}
SPL {X  -165.650, Y  +656.573, Z    +0.000, E1   +19.875, E3 +298958.626}
SPL {X  -165.650, Y  +647.335, Z    +0.000, E1   +32.835, E3 +298955.548}
SPL {X  -165.650, Y  +637.438, Z    +0.000, E1   +46.409, E3 +298950.908}
SPL {X  -165.650, Y  +605.320, Z    +0.000, E1   +76.562, E3 +298931.463}
SPL {X  -165.650, Y  +596.505, Z    +0.000, E1   +55.802, E3 +298980.819}
SPL {X  -165.650, Y  +524.050, Z    +0.000, E1   +59.300, E3 +299044.978}
ENDSPLINE

SPLINE
SPL {X  -165.650, Y  +539.856, Z    +0.000, E1   +53.398, E3 +299060.626}
ENDSPLINE

SPLINE
SPL {X  -165.650, Y  +530.389, Z    +0.000, E1   +53.621, E3 +299073.631}
SPL {X  -165.650, Y  +521.849, Z    +0.000, E1   +53.452, E3 +299087.571}
SPL {X  -165.650, Y  +515.134, Z    +0.000, E1   +53.252, E3 +299098.922}
SPL {X  -165.650, Y  +505.685, Z    +0.000, E1   +53.701, E3 +299110.529}
SPL {X  -165.650, Y  +498.275, Z    +0.000, E1   +53.357, E3 +299123.837}
SPL {X  -165.650, Y  +491.031, Z    +0.000, E1   +53.348, E3 +299134.857}
SPL {X  -165.650, Y  +479.077, Z    +0.000, E1   +55.039, E3 +299141.980}
SPL {X  -165.650, Y  +450.615, Z    +0.000, E1   +59.721, E3 +299148.486}
SPL {X  -165.650, Y  +449.326, Z    +0.000, E1   +58.606, E3 +299157.535}
SPL {X  -165.650, Y  +442.154, Z    +0.000, E1   +58.369, E3 +299168.159}
SPL {X  -165.650, Y  +437.405, Z    +0.000, E1   +57.663, E3 +299178.769}
SPL {X  -165.650, Y  +432.227, Z    +0.000, E1   +57.103, E3 +299189.256}
SPL {X  -165.650, Y  +428.683, Z    +0.000, E1   +56.222, E3 +299199.611}
SPL {X  -165.650, Y  +424.202, Z    +0.000, E1   +55.382, E3 +299211.300}
SPL {X  -165.650, Y  +418.756, Z    +0.000, E1   +54.154, E3 +299226.979}
SPL {X  -165.650, Y  +407.872, Z    +0.000, E1   +54.003, E3 +299244.064}
SPL {X  -165.650, Y  +400.791, Z    +0.000, E1   +53.827, E3 +299255.507}
SPL {X  -165.650, Y  +393.046, Z    +0.000, E1   +53.951, E3 +299266.399}
SPL {X  -165.650, Y  +383.306, Z    +0.000, E1   +53.987, E3 +299280.676}
SPL {X  -165.640, Y  +376.676, Z    +0.000, E1   +53.760, E3 +299291.843}
SPL {X  -165.408, Y  +369.556, Z    +0.000, E1   +53.942, E3 +299301.394}
SPL {X  -164.927, Y  +363.041, Z    +0.000, E1   +53.687, E3 +299312.690}
SPL {X  -164.096, Y  +355.862, Z    +0.000, E1   +53.838, E3 +299322.420}
SPL {X  -162.936, Y  +348.637, Z    +0.000, E1   +53.390, E3 +299336.136}
SPL {X  -161.218, Y  +340.437, Z    +0.000, E1   +53.207, E3 +299349.248}
SPL {X  -159.523, Y  +333.864, Z    +0.000, E1   +52.908, E3 +299360.870}
SPL {X  -157.624, Y  +327.563, Z    +0.000, E1   +52.705, E3 +299371.280}
SPL {X  -155.665, Y  +321.859, Z    +0.000, E1   +52.064, E3 +299383.453}
SPL {X  -152.682, Y  +314.249, Z    +0.000, E1   +51.841, E3 +299395.901}
SPL {X  -150.607, Y  +309.525, Z    +0.000, E1   +51.147, E3 +299406.385}
SPL {X  -142.104, Y  +293.374, Z    +0.000, E1   +55.775, E3 +299406.117}
SPL {X  -134.755, Y  +282.163, Z    +0.000, E1   +57.236, E3 +299412.385}
SPL {X  -117.053, Y  +261.289, Z    +0.000, E1   +49.815, E3 +299521.897}
ENDSPLINE

SPLINE
SPL {X  -148.836, Y  +305.783, Z    +0.000, E1   +38.029, E3 +299613.375}
SPL {X  -161.816, Y  +343.065, Z    +0.000, E1   +22.147, E3 +299604.025}
SPL {X  -164.614, Y  +360.007, Z    +0.000, E1   +13.213, E3 +299599.811}
SPL {X  -165.520, Y  +371.933, Z    +0.000, E1    +6.276, E3 +299602.565}
SPL {X  -165.650, Y  +378.704, Z    +0.000, E1    +1.700, E3 +299601.435}
SPL {X  -165.650, Y  +382.197, Z    +0.000, E1    -1.038, E3 +299600.508}
SPL {X  -165.650, Y  +386.782, Z    +0.000, E1    -5.783, E3 +299599.986}
SPL {X  -165.650, Y  +392.406, Z    +0.000, E1   -13.042, E3 +299597.883}
SPL {X  -165.650, Y  +398.038, Z    +0.000, E1   -20.113, E3 +299599.450}
SPL {X  -165.650, Y  +403.005, Z    +0.000, E1   -26.762, E3 +299598.632}
SPL {X  -165.650, Y  +415.469, Z    +0.000, E1   -43.461, E3 +299593.455}
SPL {X  -165.650, Y  +460.095, Z    +0.000, E1   -60.221, E3 +299611.717}
SPL {X  -165.650, Y  +535.749, Z    +0.000, E1   -60.559, E3 +299682.560}
ENDSPLINE

SPLINE
SPL {X  -165.650, Y  +516.750, Z    +0.000, E1   -54.244, E3 +299698.411}
ENDSPLINE

SPLINE
SPL {X  -165.650, Y  +524.345, Z    +0.000, E1   -54.115, E3 +299710.308}
SPL {X  -165.650, Y  +531.171, Z    +0.000, E1   -54.075, E3 +299720.746}
SPL {X  -165.650, Y  +538.771, Z    +0.000, E1   -53.840, E3 +299733.486}
SPL {X  -165.650, Y  +545.884, Z    +0.000, E1   -53.883, E3 +299743.791}
SPL {X  -165.650, Y  +553.081, Z    +0.000, E1   -53.834, E3 +299754.924}
SPL {X  -165.650, Y  +560.989, Z    +0.000, E1   -53.974, E3 +299765.761}
SPL {X  -165.650, Y  +568.053, Z    +0.000, E1   -54.124, E3 +299775.351}
SPL {X  -165.650, Y  +577.021, Z    +0.000, E1   -53.813, E3 +299790.850}
SPL {X  -165.650, Y  +587.996, Z    +0.000, E1   -53.969, E3 +299806.088}
SPL {X  -165.650, Y  +595.185, Z    +0.000, E1   -53.962, E3 +299816.797}
SPL {X  -165.650, Y  +602.138, Z    +0.000, E1   -53.941, E3 +299827.291}
SPL {X  -165.650, Y  +610.307, Z    +0.000, E1   -53.995, E3 +299839.139}
SPL {X  -165.650, Y  +617.878, Z    +0.000, E1   -53.838, E3 +299851.396}
SPL {X  -165.650, Y  +626.374, Z    +0.000, E1   -54.092, E3 +299862.411}
SPL {X  -165.650, Y  +632.964, Z    +0.000, E1   -53.887, E3 +299873.539}
SPL {X  -165.650, Y  +643.032, Z    +0.000, E1   -53.946, E3 +299888.283}
SPL {X  -165.650, Y  +654.069, Z    +0.000, E1   -54.108, E3 +299903.643}
SPL {X  -165.650, Y  +659.513, Z    +0.000, E1   -53.578, E3 +299914.869}
SPL {X  -165.650, Y  +667.820, Z    +0.000, E1   -53.975, E3 +299924.934}
SPL {X  -165.650, Y  +674.957, Z    +0.000, E1   -53.977, E3 +299935.447}
SPL {X  -165.574, Y  +680.515, Z    +0.000, E1   -53.820, E3 +299944.773}
SPL {X  -165.171, Y  +688.090, Z    +0.000, E1   -54.025, E3 +299954.734}
SPL {X  -164.558, Y  +694.489, Z    +0.000, E1   -53.745, E3 +299966.083}
SPL {X  -163.580, Y  +701.606, Z    +0.000, E1   -53.591, E3 +299977.516}
SPL {X  -162.702, Y  +706.614, Z    +0.000, E1   -53.230, E3 +299987.183}
SPL {X  -161.265, Y  +713.361, Z    +0.000, E1   -53.436, E3 +299995.991}
SPL {X  -159.936, Y  +718.632, Z    +0.000, E1   -52.857, E3 +300007.321}
SPL {X  -157.868, Y  +725.674, Z    +0.000, E1   -52.862, E3 +300017.662}
SPL {X  -156.314, Y  +730.327, Z    +0.000, E1   -52.199, E3 +300028.343}
SPL {X  -153.975, Y  +736.588, Z    +0.000, E1   -51.877, E3 +300039.373}
SPL {X  -151.181, Y  +743.207, Z    +0.000, E1   -51.549, E3 +300050.994}
SPL {X  -146.528, Y  +752.763, Z    +0.000, E1   -53.481, E3 +300055.171}
SPL {X  -137.775, Y  +767.467, Z    +0.000, E1   -56.912, E3 +300057.157}
SPL {X  -128.847, Y  +779.607, Z    +0.000, E1   -49.118, E3 +300132.173}
SPL {X   -94.133, Y  +811.804, Z    +0.000, E1   -53.019, E3 +300186.807}
ENDSPLINE

SPLINE
SPL {X  -134.098, Y  +772.750, Z    +0.000, E1   -45.587, E3 +300262.102}
SPL {X  -155.319, Y  +733.085, Z    +0.000, E1   -31.947, E3 +300252.979}
SPL {X  -162.077, Y  +709.719, Z    +0.000, E1   -21.590, E3 +300254.657}
SPL {X  -164.499, Y  +694.994, Z    +0.000, E1   -13.860, E3 +300255.442}
SPL {X  -165.382, Y  +684.927, Z    +0.000, E1    -7.984, E3 +300253.619}
SPL {X  -165.645, Y  +676.778, Z    +0.000, E1    -2.777, E3 +300253.341}
SPL {X  -165.650, Y  +672.938, Z    +0.000, E1    +0.157, E3 +300252.100}
SPL {X  -165.650, Y  +669.402, Z    +0.000, E1    +3.448, E3 +300251.491}
SPL {X  -165.650, Y  +663.061, Z    +0.000, E1   +11.076, E3 +300250.485}
SPL {X  -165.650, Y  +654.085, Z    +0.000, E1   +23.232, E3 +300249.593}
SPL {X  -165.650, Y  +639.700, Z    +0.000, E1   +43.326, E3 +300243.720}
SPL {X  -165.650, Y  +605.320, Z    +0.000, E1   +76.562, E3 +300223.130}
SPL {X  -165.650, Y  +596.505, Z    +0.000, E1   +55.802, E3 +300272.485}
SPL {X  -165.650, Y  +524.050, Z    +0.000, E1   +59.300, E3 +300336.645}
ENDSPLINE

SPLINE
SPL {X  -165.650, Y  +539.856, Z    +0.000, E1   +53.398, E3 +300352.292}
ENDSPLINE

SPLINE
SPL {X  -165.650, Y  +532.042, Z    +0.000, E1   +53.611, E3 +300362.764}
SPL {X  -165.650, Y  +523.239, Z    +0.000, E1   +53.520, E3 +300376.859}
SPL {X  -165.650, Y  +512.447, Z    +0.000, E1   +53.456, E3 +300393.497}
SPL {X  -165.650, Y  +503.994, Z    +0.000, E1   +53.652, E3 +300404.936}
SPL {X  -165.650, Y  +498.275, Z    +0.000, E1   +53.357, E3 +300415.504}
SPL {X  -165.650, Y  +487.031, Z    +0.000, E1   +53.931, E3 +300428.912}
SPL {X  -165.650, Y  +450.615, Z    +0.000, E1   +59.721, E3 +300440.152}
SPL {X  -165.650, Y  +449.326, Z    +0.000, E1   +58.606, E3 +300449.202}
SPL {X  -165.650, Y  +442.154, Z    +0.000, E1   +58.369, E3 +300459.826}
SPL {X  -165.650, Y  +437.405, Z    +0.000, E1   +57.663, E3 +300470.435}
SPL {X  -165.650, Y  +432.227, Z    +0.000, E1   +57.103, E3 +300480.923}
SPL {X  -165.650, Y  +428.683, Z    +0.000, E1   +56.222, E3 +300491.277}
SPL {X  -165.650, Y  +424.202, Z    +0.000, E1   +55.382, E3 +300502.966}
SPL {X  -165.650, Y  +418.756, Z    +0.000, E1   +54.154, E3 +300518.645}
SPL {X  -165.650, Y  +410.508, Z    +0.000, E1   +54.007, E3 +300531.601}
SPL {X  -165.650, Y  +403.104, Z    +0.000, E1   +53.908, E3 +300543.382}
SPL {X  -165.650, Y  +391.401, Z    +0.000, E1   +53.934, E3 +300560.773}
SPL {X  -165.650, Y  +381.191, Z    +0.000, E1   +54.078, E3 +300574.843}
SPL {X  -165.600, Y  +374.450, Z    +0.000, E1   +53.824, E3 +300586.544}
SPL {X  -165.050, Y  +364.408, Z    +0.000, E1   +53.830, E3 +300601.603}
SPL {X  -164.096, Y  +355.862, Z    +0.000, E1   +53.838, E3 +300614.087}
SPL {X  -162.936, Y  +348.637, Z    +0.000, E1   +53.390, E3 +300627.803}
SPL {X  -161.218, Y  +340.437, Z    +0.000, E1   +53.207, E3 +300640.915}
SPL {X  -159.523, Y  +333.864, Z    +0.000, E1   +52.908, E3 +300652.537}
SPL {X  -157.624, Y  +327.563, Z    +0.000, E1   +52.705, E3 +300662.946}
SPL {X  -155.665, Y  +321.859, Z    +0.000, E1   +52.064, E3 +300675.119}
SPL {X  -152.682, Y  +314.249, Z    +0.000, E1   +51.841, E3 +300687.567}
SPL {X  -150.607, Y  +309.525, Z    +0.000, E1   +51.147, E3 +300698.052}
SPL {X  -142.104, Y  +293.374, Z    +0.000, E1   +55.775, E3 +300697.784}
SPL {X  -134.755, Y  +282.163, Z    +0.000, E1   +57.236, E3 +300704.052}
SPL {X  -117.053, Y  +261.289, Z    +0.000, E1   +49.815, E3 +300813.564}
ENDSPLINE

SPLINE
SPL {X  -148.836, Y  +305.783, Z    +0.000, E1   +38.029, E3 +300905.041}
SPL {X  -161.816, Y  +343.065, Z    +0.000, E1   +22.147, E3 +300895.691}
SPL {X  -165.007, Y  +363.921, Z    +0.000, E1   +11.079, E3 +300893.680}
SPL {X  -165.587, Y  +373.939, Z    +0.000, E1    +4.928, E3 +300893.520}
SPL {X  -165.650, Y  +380.164, Z    +0.000, E1    +0.707, E3 +300892.701}
SPL {X  -165.650, Y  +383.228, Z    +0.000, E1    -2.108, E3 +300891.926}
SPL {X  -165.650, Y  +386.782, Z    +0.000, E1    -5.783, E3 +300891.652}
SPL {X  -165.650, Y  +392.406, Z    +0.000, E1   -13.042, E3 +300889.550}
SPL {X  -165.650, Y  +398.038, Z    +0.000, E1   -20.113, E3 +300891.117}
SPL {X  -165.650, Y  +403.005, Z    +0.000, E1   -26.762, E3 +300890.299}
SPL {X  -165.650, Y  +415.469, Z    +0.000, E1   -43.461, E3 +300885.122}
SPL {X  -165.650, Y  +460.095, Z    +0.000, E1   -60.221, E3 +300903.383}
SPL {X  -165.650, Y  +535.749, Z    +0.000, E1   -60.559, E3 +300974.227}
ENDSPLINE

SPLINE
SPL {X  -165.650, Y  +516.750, Z    +0.000, E1   -54.244, E3 +300990.077}
ENDSPLINE

SPLINE
SPL {X  -165.650, Y  +524.345, Z    +0.000, E1   -54.115, E3 +301001.974}
SPL {X  -165.650, Y  +531.171, Z    +0.000, E1   -54.075, E3 +301012.413}
SPL {X  -165.650, Y  +538.771, Z    +0.000, E1   -53.840, E3 +301025.153}
SPL {X  -165.650, Y  +548.103, Z    +0.000, E1   -53.944, E3 +301038.500}
SPL {X  -165.650, Y  +558.071, Z    +0.000, E1   -53.870, E3 +301053.840}
SPL {X  -165.650, Y  +568.053, Z    +0.000, E1   -54.124, E3 +301067.018}
SPL {X  -165.650, Y  +577.021, Z    +0.000, E1   -53.813, E3 +301082.517}
SPL {X  -165.650, Y  +587.996, Z    +0.000, E1   -53.969, E3 +301097.754}
SPL {X  -165.650, Y  +595.185, Z    +0.000, E1   -53.962, E3 +301108.464}
SPL {X  -165.650, Y  +602.138, Z    +0.000, E1   -53.941, E3 +301118.958}
SPL {X  -165.650, Y  +610.307, Z    +0.000, E1   -53.995, E3 +301130.806}
SPL {X  -165.650, Y  +617.878, Z    +0.000, E1   -53.838, E3 +301143.062}
SPL {X  -165.650, Y  +626.374, Z    +0.000, E1   -54.092, E3 +301154.078}
SPL {X  -165.650, Y  +632.964, Z    +0.000, E1   -53.887, E3 +301165.205}
SPL {X  -165.650, Y  +643.032, Z    +0.000, E1   -53.946, E3 +301179.950}
SPL {X  -165.650, Y  +654.069, Z    +0.000, E1   -54.108, E3 +301195.309}
SPL {X  -165.650, Y  +659.513, Z    +0.000, E1   -53.578, E3 +301206.536}
SPL {X  -165.650, Y  +667.820, Z    +0.000, E1   -53.975, E3 +301216.601}
SPL {X  -165.623, Y  +678.503, Z    +0.000, E1   -53.932, E3 +301232.953}
SPL {X  -165.027, Y  +689.850, Z    +0.000, E1   -53.862, E3 +301250.216}
SPL {X  -163.840, Y  +699.919, Z    +0.000, E1   -53.732, E3 +301265.998}
SPL {X  -162.702, Y  +706.614, Z    +0.000, E1   -53.230, E3 +301278.849}
SPL {X  -161.265, Y  +713.361, Z    +0.000, E1   -53.436, E3 +301287.658}
SPL {X  -159.936, Y  +718.632, Z    +0.000, E1   -52.857, E3 +301298.987}
SPL {X  -157.868, Y  +725.674, Z    +0.000, E1   -52.862, E3 +301309.328}
SPL {X  -156.314, Y  +730.327, Z    +0.000, E1   -52.199, E3 +301320.010}
SPL {X  -153.975, Y  +736.588, Z    +0.000, E1   -51.877, E3 +301331.040}
SPL {X  -151.949, Y  +741.465, Z    +0.000, E1   -51.645, E3 +301339.445}
SPL {X  -149.075, Y  +747.727, Z    +0.000, E1   -52.134, E3 +301346.160}
SPL {X  -137.775, Y  +767.467, Z    +0.000, E1   -56.912, E3 +301348.823}
SPL {X  -128.847, Y  +779.607, Z    +0.000, E1   -49.118, E3 +301423.840}
SPL {X   -94.133, Y  +811.804, Z    +0.000, E1   -53.019, E3 +301478.474}
ENDSPLINE

SPLINE
SPL {X  -134.098, Y  +772.750, Z    +0.000, E1   -45.587, E3 +301553.768}
SPL {X  -155.319, Y  +733.085, Z    +0.000, E1   -31.947, E3 +301544.646}
SPL {X  -162.077, Y  +709.719, Z    +0.000, E1   -21.590, E3 +301546.324}
SPL {X  -164.499, Y  +694.994, Z    +0.000, E1   -13.860, E3 +301547.108}
SPL {X  -165.513, Y  +682.236, Z    +0.000, E1    -6.385, E3 +301545.444}
SPL {X  -165.650, Y  +675.776, Z    +0.000, E1    -2.014, E3 +301544.752}
SPL {X  -165.650, Y  +672.938, Z    +0.000, E1    +0.157, E3 +301543.767}
SPL {X  -165.650, Y  +669.402, Z    +0.000, E1    +3.448, E3 +301543.158}
SPL {X  -165.650, Y  +663.061, Z    +0.000, E1   +11.076, E3 +301542.152}
SPL {X  -165.650, Y  +656.573, Z    +0.000, E1   +19.875, E3 +301541.959}
SPL {X  -165.650, Y  +650.769, Z    +0.000, E1   +28.083, E3 +301540.325}
SPL {X  -165.650, Y  +639.700, Z    +0.000, E1   +43.326, E3 +301535.387}
SPL {X  -165.650, Y  +605.320, Z    +0.000, E1   +76.562, E3 +301514.796}
SPL {X  -165.650, Y  +597.745, Z    +0.000, E1   +59.636, E3 +301552.798}
SPL {X  -165.650, Y  +596.360, Z    +0.000, E1   +54.978, E3 +301566.406}
SPL {X  -165.650, Y  +521.429, Z    +0.000, E1   +61.144, E3 +301619.637}
ENDSPLINE

SPLINE
SPL {X  -165.650, Y  +526.028, Z    +0.000, E1   +58.071, E3 +301633.411}
SPL {X  -165.650, Y  +539.856, Z    +0.000, E1   +53.398, E3 +301643.959}
ENDSPLINE

SPLINE
SPL {X  -165.650, Y  +532.042, Z    +0.000, E1   +53.611, E3 +301654.430}
SPL {X  -165.650, Y  +526.147, Z    +0.000, E1   +53.495, E3 +301664.069}
SPL {X  -165.650, Y  +517.365, Z    +0.000, E1   +53.387, E3 +301678.237}
SPL {X  -165.650, Y  +505.685, Z    +0.000, E1   +53.701, E3 +301693.863}
SPL {X  -165.650, Y  +498.275, Z    +0.000, E1   +53.357, E3 +301707.170}
SPL {X  -165.650, Y  +487.031, Z    +0.000, E1   +53.931, E3 +301720.579}
SPL {X  -165.650, Y  +450.615, Z    +0.000, E1   +59.721, E3 +301731.819}
SPL {X  -165.650, Y  +449.326, Z    +0.000, E1   +58.606, E3 +301740.868}
SPL {X  -165.650, Y  +442.154, Z    +0.000, E1   +58.369, E3 +301751.492}
SPL {X  -165.650, Y  +437.405, Z    +0.000, E1   +57.663, E3 +301762.102}
SPL {X  -165.650, Y  +432.227, Z    +0.000, E1   +57.103, E3 +301772.590}
SPL {X  -165.650, Y  +428.683, Z    +0.000, E1   +56.222, E3 +301782.944}
SPL {X  -165.650, Y  +424.202, Z    +0.000, E1   +55.382, E3 +301794.633}
SPL {X  -165.650, Y  +418.756, Z    +0.000, E1   +54.154, E3 +301810.312}
SPL {X  -165.650, Y  +410.508, Z    +0.000, E1   +54.007, E3 +301823.267}
SPL {X  -165.650, Y  +403.104, Z    +0.000, E1   +53.908, E3 +301835.049}
SPL {X  -165.650, Y  +393.046, Z    +0.000, E1   +53.951, E3 +301849.732}
SPL {X  -165.650, Y  +383.306, Z    +0.000, E1   +53.987, E3 +301864.010}
SPL {X  -165.640, Y  +376.676, Z    +0.000, E1   +53.760, E3 +301875.176}
SPL {X  -165.408, Y  +369.556, Z    +0.000, E1   +53.942, E3 +301884.727}
SPL {X  -164.927, Y  +363.041, Z    +0.000, E1   +53.687, E3 +301896.023}
SPL {X  -163.980, Y  +355.035, Z    +0.000, E1   +53.657, E3 +301908.219}
SPL {X  -162.665, Y  +347.197, Z    +0.000, E1   +53.396, E3 +301921.483}
SPL {X  -161.218, Y  +340.437, Z    +0.000, E1   +53.207, E3 +301932.581}
SPL {X  -159.523, Y  +333.864, Z    +0.000, E1   +52.908, E3 +301944.204}
SPL {X  -157.624, Y  +327.563, Z    +0.000, E1   +52.705, E3 +301954.613}
SPL {X  -156.289, Y  +323.602, Z    +0.000, E1   +52.159, E3 +301963.502}
SPL {X  -153.877, Y  +317.168, Z    +0.000, E1   +51.945, E3 +301974.363}
SPL {X  -151.035, Y  +310.467, Z    +0.000, E1   +51.312, E3 +301987.608}
SPL {X  -139.567, Y  +289.276, Z    +0.000, E1   +56.334, E3 +301991.697}
SPL {X  -117.053, Y  +261.289, Z    +0.000, E1   +49.815, E3 +302105.230}
ENDSPLINE

SPLINE
SPL {X  -148.836, Y  +305.783, Z    +0.000, E1   +38.029, E3 +302196.708}
SPL {X  -161.816, Y  +343.065, Z    +0.000, E1   +22.147, E3 +302187.358}
SPL {X  -164.614, Y  +360.007, Z    +0.000, E1   +13.213, E3 +302183.144}
SPL {X  -165.520, Y  +371.933, Z    +0.000, E1    +6.276, E3 +302185.899}
SPL {X  -165.650, Y  +378.704, Z    +0.000, E1    +1.700, E3 +302184.768}
SPL {X  -165.650, Y  +382.197, Z    +0.000, E1    -1.038, E3 +302183.841}
SPL {X  -165.650, Y  +386.782, Z    +0.000, E1    -5.783, E3 +302183.319}
SPL {X  -165.650, Y  +392.406, Z    +0.000, E1   -13.042, E3 +302181.216}
SPL {X  -165.650, Y  +400.489, Z    +0.000, E1   -23.243, E3 +302182.380}
SPL {X  -165.650, Y  +415.469, Z    +0.000, E1   -43.461, E3 +302176.789}
SPL {X  -165.650, Y  +460.095, Z    +0.000, E1   -60.221, E3 +302195.050}
SPL {X  -165.650, Y  +535.749, Z    +0.000, E1   -60.559, E3 +302265.894}
ENDSPLINE

SPLINE
SPL {X  -165.650, Y  +516.866, Z    +0.000, E1   -54.768, E3 +302278.444}
ENDSPLINE

SPLINE
SPL {X  -165.650, Y  +521.328, Z    +0.000, E1   -53.870, E3 +302290.735}
SPL {X  -165.650, Y  +531.171, Z    +0.000, E1   -54.075, E3 +302304.079}
SPL {X  -165.650, Y  +538.771, Z    +0.000, E1   -53.840, E3 +302316.820}
SPL {X  -165.650, Y  +548.103, Z    +0.000, E1   -53.944, E3 +302330.166}
SPL {X  -165.650, Y  +558.071, Z    +0.000, E1   -53.870, E3 +302345.507}
SPL {X  -165.650, Y  +568.053, Z    +0.000, E1   -54.124, E3 +302358.685}
SPL {X  -165.650, Y  +577.021, Z    +0.000, E1   -53.813, E3 +302374.183}
SPL {X  -165.650, Y  +587.996, Z    +0.000, E1   -53.969, E3 +302389.421}
SPL {X  -165.650, Y  +595.185, Z    +0.000, E1   -53.962, E3 +302400.130}
SPL {X  -165.650, Y  +602.138, Z    +0.000, E1   -53.941, E3 +302410.625}
SPL {X  -165.650, Y  +610.307, Z    +0.000, E1   -53.995, E3 +302422.472}
SPL {X  -165.650, Y  +617.878, Z    +0.000, E1   -53.838, E3 +302434.729}
SPL {X  -165.650, Y  +627.853, Z    +0.000, E1   -53.937, E3 +302449.083}
SPL {X  -165.650, Y  +638.510, Z    +0.000, E1   -54.057, E3 +302464.142}
SPL {X  -165.650, Y  +647.911, Z    +0.000, E1   -53.930, E3 +302478.941}
SPL {X  -165.650, Y  +658.189, Z    +0.000, E1   -53.932, E3 +302494.241}
SPL {X  -165.650, Y  +667.820, Z    +0.000, E1   -53.975, E3 +302508.268}
SPL {X  -165.623, Y  +678.503, Z    +0.000, E1   -53.932, E3 +302524.619}
SPL {X  -165.171, Y  +688.090, Z    +0.000, E1   -54.025, E3 +302538.067}
SPL {X  -164.558, Y  +694.489, Z    +0.000, E1   -53.745, E3 +302549.416}
SPL {X  -163.580, Y  +701.606, Z    +0.000, E1   -53.591, E3 +302560.849}
SPL {X  -162.702, Y  +706.614, Z    +0.000, E1   -53.230, E3 +302570.516}
SPL {X  -160.941, Y  +714.715, Z    +0.000, E1   -53.321, E3 +302582.136}
SPL {X  -159.638, Y  +719.723, Z    +0.000, E1   -52.685, E3 +302593.138}
SPL {X  -157.521, Y  +726.754, Z    +0.000, E1   -52.585, E3 +302604.334}
SPL {X  -155.632, Y  +732.234, Z    +0.000, E1   -52.209, E3 +302614.380}
SPL {X  -153.975, Y  +736.588, Z    +0.000, E1   -51.877, E3 +302622.707}
SPL {X  -151.949, Y  +741.465, Z    +0.000, E1   -51.645, E3 +302631.112}
SPL {X  -149.075, Y  +747.727, Z    +0.000, E1   -52.134, E3 +302637.827}
SPL {X  -137.775, Y  +767.467, Z    +0.000, E1   -56.912, E3 +302640.490}
SPL {X  -128.847, Y  +779.607, Z    +0.000, E1   -49.118, E3 +302715.506}
SPL {X   -94.133, Y  +811.804, Z    +0.000, E1   -53.019, E3 +302770.141}
ENDSPLINE

